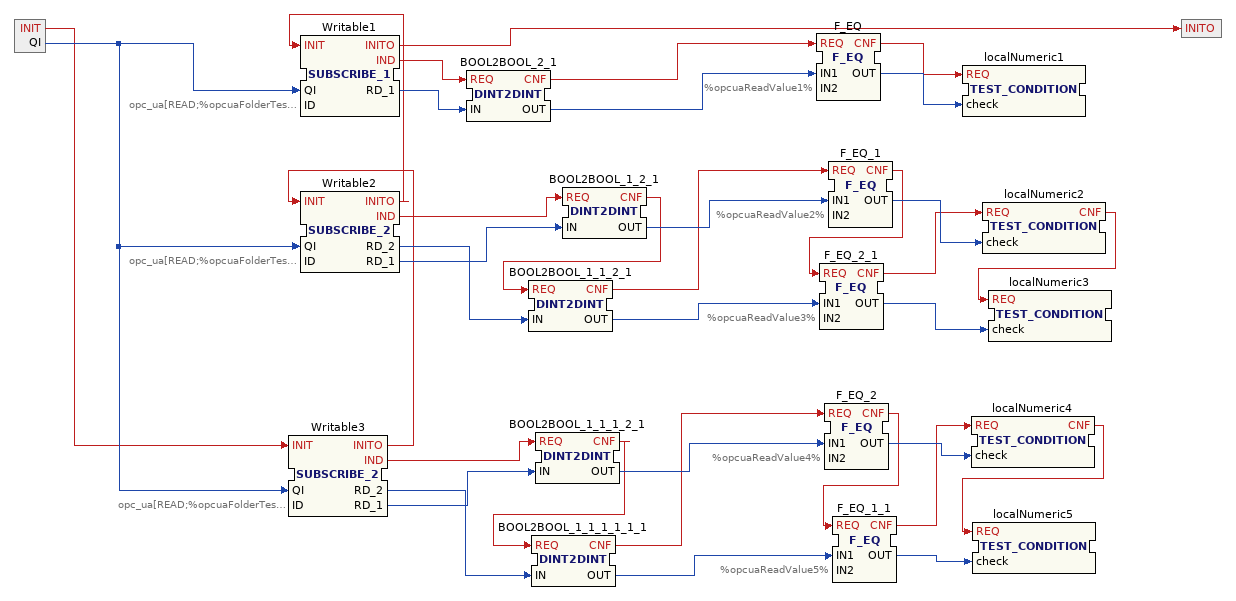
      [picture p121: application OpcUADelayedWorking.numericNodeIdTest]
      FBS
        BOOL2BOOL_1_2_1 : DINT2DINT;
        BOOL2BOOL_2_1 : DINT2DINT;
        BOOL2BOOL_1_1_2_1 : DINT2DINT;
        BOOL2BOOL_1_1_1_2_1 : DINT2DINT;
        BOOL2BOOL_1_1_1_1_1_1 : DINT2DINT;
        Writable1 : SUBSCRIBE_1(ID := opc_ua[READ;%opcuaFolderTestWithNodeIdNumeric1%]);
        Writable2 : SUBSCRIBE_2(ID := opc_ua[READ;%opcuaFolderTestWithNodeIdNumeric2%]);
        Writable3 : SUBSCRIBE_2(ID := opc_ua[READ;%opcuaFolderTestWithNodeIdNumeric3%]);
        localNumeric1 : TEST_CONDITION;
        localNumeric2 : TEST_CONDITION;
        localNumeric3 : TEST_CONDITION;
        localNumeric4 : TEST_CONDITION;
        localNumeric5 : TEST_CONDITION;
        F_EQ : F_EQ(IN2 := %opcuaReadValue1%);
        F_EQ_1 : F_EQ(IN2 := %opcuaReadValue2%);
        F_EQ_2 : F_EQ(IN2 := %opcuaReadValue4%);
        F_EQ_1_1 : F_EQ(IN2 := %opcuaReadValue5%);
        F_EQ_2_1 : F_EQ(IN2 := %opcuaReadValue3%);
      END_FBS
      EVENT_CONNECTIONS
        Writable1.INITO TO INITO;
        Writable2.INITO TO Writable1.INIT;
        INIT TO Writable3.INIT;
        Writable3.INITO TO Writable2.INIT;
        Writable1.IND TO BOOL2BOOL_2_1.REQ;
        Writable2.IND TO BOOL2BOOL_1_2_1.REQ;
        BOOL2BOOL_1_2_1.CNF TO BOOL2BOOL_1_1_2_1.REQ;
        Writable3.IND TO BOOL2BOOL_1_1_1_2_1.REQ;
        BOOL2BOOL_1_1_1_2_1.CNF TO BOOL2BOOL_1_1_1_1_1_1.REQ;
        BOOL2BOOL_2_1.CNF TO F_EQ.REQ;
        F_EQ.CNF TO localNumeric1.REQ;
        BOOL2BOOL_1_1_2_1.CNF TO F_EQ_1.REQ;
        F_EQ_1.CNF TO F_EQ_2_1.REQ;
        F_EQ_2_1.CNF TO localNumeric2.REQ;
        BOOL2BOOL_1_1_1_1_1_1.CNF TO F_EQ_2.REQ;
        F_EQ_2.CNF TO F_EQ_1_1.REQ;
        F_EQ_1_1.CNF TO localNumeric4.REQ;
        localNumeric4.CNF TO localNumeric5.REQ;
        localNumeric2.CNF TO localNumeric3.REQ;
      END_CONNECTIONS
      DATA_CONNECTIONS
        QI TO Writable1.QI;
        QI TO Writable2.QI;
        QI TO Writable3.QI;
        Writable1.RD_1 TO BOOL2BOOL_2_1.IN;
        Writable3.RD_2 TO BOOL2BOOL_1_1_1_1_1_1.IN;
        Writable3.RD_1 TO BOOL2BOOL_1_1_1_2_1.IN;
        Writable2.RD_2 TO BOOL2BOOL_1_1_2_1.IN;
        Writable2.RD_1 TO BOOL2BOOL_1_2_1.IN;
        BOOL2BOOL_2_1.OUT TO F_EQ.IN1;
        F_EQ.OUT TO localNumeric1.check;
        BOOL2BOOL_1_1_2_1.OUT TO F_EQ_2_1.IN1;
        BOOL2BOOL_1_2_1.OUT TO F_EQ_1.IN1;
        BOOL2BOOL_1_1_1_2_1.OUT TO F_EQ_2.IN1;
        BOOL2BOOL_1_1_1_1_1_1.OUT TO F_EQ_1_1.IN1;
        F_EQ_1_1.OUT TO localNumeric5.check;
        F_EQ_2.OUT TO localNumeric4.check;
        F_EQ_2_1.OUT TO localNumeric3.check;
        F_EQ_1.OUT TO localNumeric2.check;
      END_CONNECTIONS
    END_SUBAPPLICATION
    SUBAPPLICATION folderTest
      EVENT_INPUT
        INIT;
      END_EVENT
      EVENT_OUTPUT
        INITO;
      END_EVENT
      VAR_INPUT
        QI : BOOL;
      END_VAR
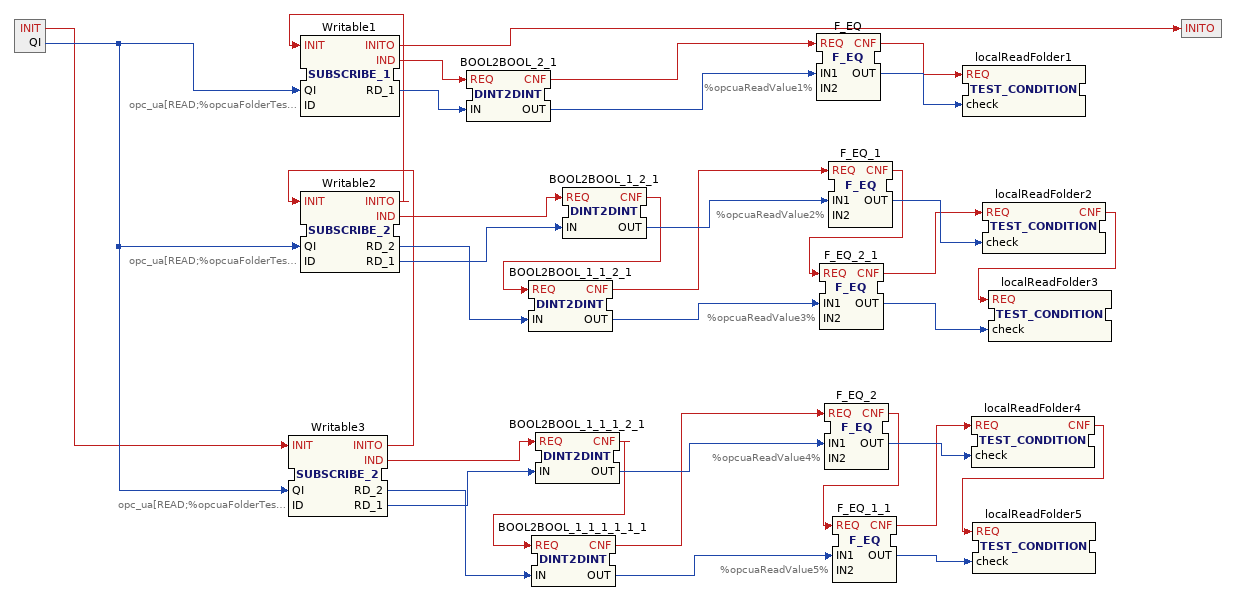
      FBS
        BOOL2BOOL_1_2_1 : DINT2DINT;
        BOOL2BOOL_2_1 : DINT2DINT;
        BOOL2BOOL_1_1_2_1 : DINT2DINT;
        BOOL2BOOL_1_1_1_2_1 : DINT2DINT;
        BOOL2BOOL_1_1_1_1_1_1 : DINT2DINT;
        Writable1 : SUBSCRIBE_1(ID := opc_ua[READ;%opcuaFolderTestOnlyBroseName1%]);
        Writable2 : SUBSCRIBE_2(ID := opc_ua[READ;%opcuaFolderTestOnlyBroseName2%]);
        Writable3 : SUBSCRIBE_2(ID := opc_ua[READ;%opcuaFolderTestOnlyBroseName3%]);
        localReadFolder1 : TEST_CONDITION;
        localReadFolder2 : TEST_CONDITION;
        localReadFolder3 : TEST_CONDITION;
        localReadFolder4 : TEST_CONDITION;
        localReadFolder5 : TEST_CONDITION;
        F_EQ : F_EQ(IN2 := %opcuaReadValue1%);
        F_EQ_1 : F_EQ(IN2 := %opcuaReadValue2%);
        F_EQ_2 : F_EQ(IN2 := %opcuaReadValue4%);
        F_EQ_1_1 : F_EQ(IN2 := %opcuaReadValue5%);
        F_EQ_2_1 : F_EQ(IN2 := %opcuaReadValue3%);
      END_FBS
      EVENT_CONNECTIONS
        Writable1.INITO TO INITO;
        Writable2.INITO TO Writable1.INIT;
        INIT TO Writable3.INIT;
        Writable3.INITO TO Writable2.INIT;
        Writable1.IND TO BOOL2BOOL_2_1.REQ;
        Writable2.IND TO BOOL2BOOL_1_2_1.REQ;
        BOOL2BOOL_1_2_1.CNF TO BOOL2BOOL_1_1_2_1.REQ;
        Writable3.IND TO BOOL2BOOL_1_1_1_2_1.REQ;
        BOOL2BOOL_1_1_1_2_1.CNF TO BOOL2BOOL_1_1_1_1_1_1.REQ;
        BOOL2BOOL_2_1.CNF TO F_EQ.REQ;
        F_EQ.CNF TO localReadFolder1.REQ;
        BOOL2BOOL_1_1_2_1.CNF TO F_EQ_1.REQ;
        F_EQ_1.CNF TO F_EQ_2_1.REQ;
        F_EQ_2_1.CNF TO localReadFolder2.REQ;
        BOOL2BOOL_1_1_1_1_1_1.CNF TO F_EQ_2.REQ;
        F_EQ_2.CNF TO F_EQ_1_1.REQ;
        F_EQ_1_1.CNF TO localReadFolder4.REQ;
        localReadFolder4.CNF TO localReadFolder5.REQ;
        localReadFolder2.CNF TO localReadFolder3.REQ;
      END_CONNECTIONS
      DATA_CONNECTIONS
        QI TO Writable1.QI;
        QI TO Writable2.QI;
        QI TO Writable3.QI;
        Writable1.RD_1 TO BOOL2BOOL_2_1.IN;
        Writable3.RD_2 TO BOOL2BOOL_1_1_1_1_1_1.IN;
        Writable3.RD_1 TO BOOL2BOOL_1_1_1_2_1.IN;
        Writable2.RD_2 TO BOOL2BOOL_1_1_2_1.IN;
        Writable2.RD_1 TO BOOL2BOOL_1_2_1.IN;
        BOOL2BOOL_2_1.OUT TO F_EQ.IN1;
        F_EQ.OUT TO localReadFolder1.check;
        BOOL2BOOL_1_1_2_1.OUT TO F_EQ_2_1.IN1;
        BOOL2BOOL_1_2_1.OUT TO F_EQ_1.IN1;
        BOOL2BOOL_1_1_1_2_1.OUT TO F_EQ_2.IN1;
        BOOL2BOOL_1_1_1_1_1_1.OUT TO F_EQ_1_1.IN1;
        F_EQ_1_1.OUT TO localReadFolder5.check;
        F_EQ_2.OUT TO localReadFolder4.check;
        F_EQ_2_1.OUT TO localReadFolder3.check;
        F_EQ_1.OUT TO localReadFolder2.check;
      END_CONNECTIONS
    END_SUBAPPLICATION
    SUBAPPLICATION byteStringNodeIdTest
      EVENT_INPUT
        INIT;
      END_EVENT
      EVENT_OUTPUT
        INITO;
      END_EVENT
      VAR_INPUT
        QI : BOOL;
      END_VAR
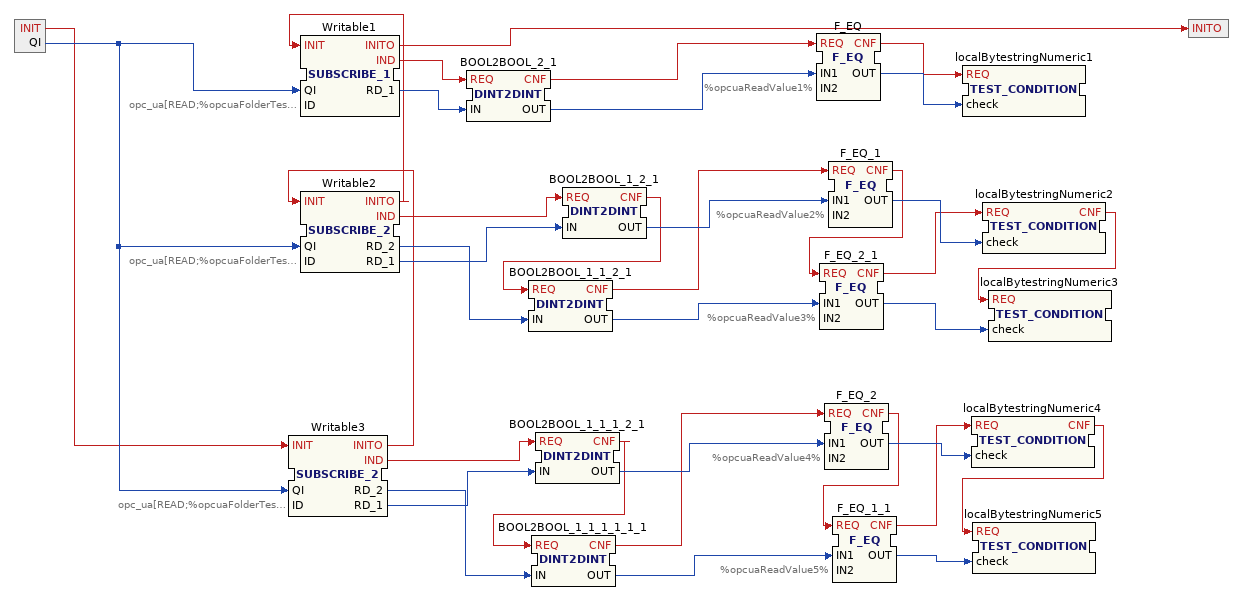
      FBS
        BOOL2BOOL_1_2_1 : DINT2DINT;
        BOOL2BOOL_2_1 : DINT2DINT;
        BOOL2BOOL_1_1_2_1 : DINT2DINT;
        BOOL2BOOL_1_1_1_2_1 : DINT2DINT;
        BOOL2BOOL_1_1_1_1_1_1 : DINT2DINT;
        Writable1 : SUBSCRIBE_1(ID := opc_ua[READ;%opcuaFolderTestWithNodeIdByteString1%]);
        Writable2 : SUBSCRIBE_2(ID := opc_ua[READ;%opcuaFolderTestWithNodeIdByteString2%]);
        Writable3 : SUBSCRIBE_2(ID := opc_ua[READ;%opcuaFolderTestWithNodeIdByteString3%]);
        localBytestringNumeric1 : TEST_CONDITION;
        localBytestringNumeric2 : TEST_CONDITION;
        localBytestringNumeric3 : TEST_CONDITION;
        localBytestringNumeric4 : TEST_CONDITION;
        localBytestringNumeric5 : TEST_CONDITION;
        F_EQ : F_EQ(IN2 := %opcuaReadValue1%);
        F_EQ_1 : F_EQ(IN2 := %opcuaReadValue2%);
        F_EQ_2 : F_EQ(IN2 := %opcuaReadValue4%);
        F_EQ_1_1 : F_EQ(IN2 := %opcuaReadValue5%);
        F_EQ_2_1 : F_EQ(IN2 := %opcuaReadValue3%);
      END_FBS
      EVENT_CONNECTIONS
        Writable1.INITO TO INITO;
        Writable2.INITO TO Writable1.INIT;
        INIT TO Writable3.INIT;
        Writable3.INITO TO Writable2.INIT;
        Writable1.IND TO BOOL2BOOL_2_1.REQ;
        Writable2.IND TO BOOL2BOOL_1_2_1.REQ;
        BOOL2BOOL_1_2_1.CNF TO BOOL2BOOL_1_1_2_1.REQ;
        Writable3.IND TO BOOL2BOOL_1_1_1_2_1.REQ;
        BOOL2BOOL_1_1_1_2_1.CNF TO BOOL2BOOL_1_1_1_1_1_1.REQ;
        BOOL2BOOL_2_1.CNF TO F_EQ.REQ;
        F_EQ.CNF TO localBytestringNumeric1.REQ;
        BOOL2BOOL_1_1_2_1.CNF TO F_EQ_1.REQ;
        F_EQ_1.CNF TO F_EQ_2_1.REQ;
        F_EQ_2_1.CNF TO localBytestringNumeric2.REQ;
        BOOL2BOOL_1_1_1_1_1_1.CNF TO F_EQ_2.REQ;
        F_EQ_2.CNF TO F_EQ_1_1.REQ;
        F_EQ_1_1.CNF TO localBytestringNumeric4.REQ;
        localBytestringNumeric4.CNF TO localBytestringNumeric5.REQ;
        localBytestringNumeric2.CNF TO localBytestringNumeric3.REQ;
      END_CONNECTIONS
      DATA_CONNECTIONS
        QI TO Writable1.QI;
        QI TO Writable2.QI;
        QI TO Writable3.QI;
        Writable1.RD_1 TO BOOL2BOOL_2_1.IN;
        Writable3.RD_2 TO BOOL2BOOL_1_1_1_1_1_1.IN;
        Writable3.RD_1 TO BOOL2BOOL_1_1_1_2_1.IN;
        Writable2.RD_2 TO BOOL2BOOL_1_1_2_1.IN;
        Writable2.RD_1 TO BOOL2BOOL_1_2_1.IN;
        BOOL2BOOL_2_1.OUT TO F_EQ.IN1;
        F_EQ.OUT TO localBytestringNumeric1.check;
        BOOL2BOOL_1_1_2_1.OUT TO F_EQ_2_1.IN1;
        BOOL2BOOL_1_2_1.OUT TO F_EQ_1.IN1;
        BOOL2BOOL_1_1_1_2_1.OUT TO F_EQ_2.IN1;
        BOOL2BOOL_1_1_1_1_1_1.OUT TO F_EQ_1_1.IN1;
        F_EQ_1_1.OUT TO localBytestringNumeric5.check;
        F_EQ_2.OUT TO localBytestringNumeric4.check;
        F_EQ_2_1.OUT TO localBytestringNumeric3.check;
        F_EQ_1.OUT TO localBytestringNumeric2.check;
      END_CONNECTIONS
    END_SUBAPPLICATION
    SUBAPPLICATION stringNodeIdTestt
      EVENT_INPUT
        INIT;
      END_EVENT
      EVENT_OUTPUT
        INITO;
      END_EVENT
      VAR_INPUT
        QI : BOOL;
      END_VAR
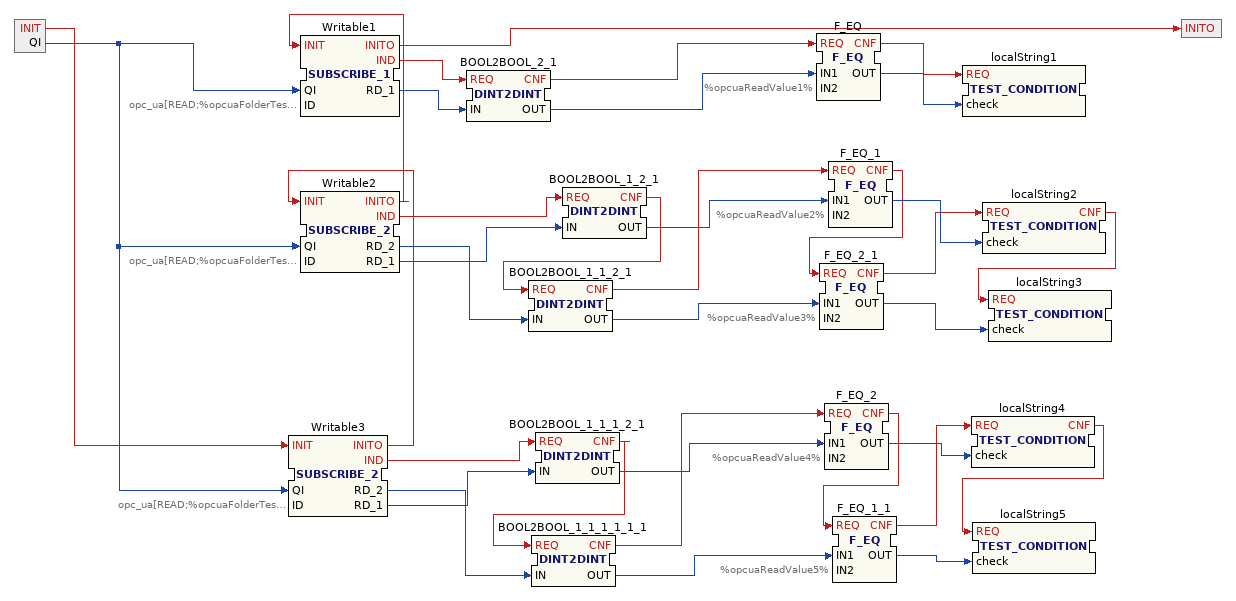
      FBS
        BOOL2BOOL_1_2_1 : DINT2DINT;
        BOOL2BOOL_2_1 : DINT2DINT;
        BOOL2BOOL_1_1_2_1 : DINT2DINT;
        BOOL2BOOL_1_1_1_2_1 : DINT2DINT;
        BOOL2BOOL_1_1_1_1_1_1 : DINT2DINT;
        Writable1 : SUBSCRIBE_1(ID := opc_ua[READ;%opcuaFolderTestWithNodeIdString1%]);
        Writable2 : SUBSCRIBE_2(ID := opc_ua[READ;%opcuaFolderTestWithNodeIdString2%]);
        Writable3 : SUBSCRIBE_2(ID := opc_ua[READ;%opcuaFolderTestWithNodeIdString3%]);
        localString1 : TEST_CONDITION;
        localString2 : TEST_CONDITION;
        localString3 : TEST_CONDITION;
        localString4 : TEST_CONDITION;
        localString5 : TEST_CONDITION;
        F_EQ : F_EQ(IN2 := %opcuaReadValue1%);
        F_EQ_1 : F_EQ(IN2 := %opcuaReadValue2%);
        F_EQ_2 : F_EQ(IN2 := %opcuaReadValue4%);
        F_EQ_1_1 : F_EQ(IN2 := %opcuaReadValue5%);
        F_EQ_2_1 : F_EQ(IN2 := %opcuaReadValue3%);
      END_FBS
      EVENT_CONNECTIONS
        Writable1.INITO TO INITO;
        Writable2.INITO TO Writable1.INIT;
        INIT TO Writable3.INIT;
        Writable3.INITO TO Writable2.INIT;
        Writable1.IND TO BOOL2BOOL_2_1.REQ;
        Writable2.IND TO BOOL2BOOL_1_2_1.REQ;
        BOOL2BOOL_1_2_1.CNF TO BOOL2BOOL_1_1_2_1.REQ;
        Writable3.IND TO BOOL2BOOL_1_1_1_2_1.REQ;
        BOOL2BOOL_1_1_1_2_1.CNF TO BOOL2BOOL_1_1_1_1_1_1.REQ;
        BOOL2BOOL_2_1.CNF TO F_EQ.REQ;
        F_EQ.CNF TO localString1.REQ;
        BOOL2BOOL_1_1_2_1.CNF TO F_EQ_1.REQ;
        F_EQ_1.CNF TO F_EQ_2_1.REQ;
        F_EQ_2_1.CNF TO localString2.REQ;
        BOOL2BOOL_1_1_1_1_1_1.CNF TO F_EQ_2.REQ;
        F_EQ_2.CNF TO F_EQ_1_1.REQ;
        F_EQ_1_1.CNF TO localString4.REQ;
        localString4.CNF TO localString5.REQ;
        localString2.CNF TO localString3.REQ;
      END_CONNECTIONS
      DATA_CONNECTIONS
        QI TO Writable1.QI;
        QI TO Writable2.QI;
        QI TO Writable3.QI;
        Writable1.RD_1 TO BOOL2BOOL_2_1.IN;
        Writable3.RD_2 TO BOOL2BOOL_1_1_1_1_1_1.IN;
        Writable3.RD_1 TO BOOL2BOOL_1_1_1_2_1.IN;
        Writable2.RD_2 TO BOOL2BOOL_1_1_2_1.IN;
        Writable2.RD_1 TO BOOL2BOOL_1_2_1.IN;
        BOOL2BOOL_2_1.OUT TO F_EQ.IN1;
        F_EQ.OUT TO localString1.check;
        BOOL2BOOL_1_1_2_1.OUT TO F_EQ_2_1.IN1;
        BOOL2BOOL_1_2_1.OUT TO F_EQ_1.IN1;
        BOOL2BOOL_1_1_1_2_1.OUT TO F_EQ_2.IN1;
        BOOL2BOOL_1_1_1_1_1_1.OUT TO F_EQ_1_1.IN1;
        F_EQ_1_1.OUT TO localString5.check;
        F_EQ_2.OUT TO localString4.check;
        F_EQ_2_1.OUT TO localString3.check;
        F_EQ_1.OUT TO localString2.check;
      END_CONNECTIONS
    END_SUBAPPLICATION
    EVENT_CONNECTIONS
      bytestringNodeIdTestRemote.INITO TO RemoteMethods.INIT;
      RemoteMethods.INITO TO HandleInit.InitFinished;
      folderTestRemote.CNF TO numericNodeIdTestRemote.REQ;
      HandleInit.Execute TO E_DELAY.START;
      SUBSCRIBE_0_1.IND TO E_SR.R;
      E_PERMIT.EO TO E_SR_1.S;
      numericNodeIdTestRemote.INITO TO stringNodeIdTestRemote.INIT;
      InitFinishedSignal.IND TO PUBLISH_0.REQ;
      E_DELAY.EO TO folderTestRemote.REQ;
      stringNodeIdTestRemote.INITO TO bytestringNodeIdTestRemote.INIT;
      bytestringNodeIdTestRemote.CNF TO RemoteMethods.REQ;
      folderTestRemote.INITO TO numericNodeIdTestRemote.INIT;
      InitFinishedSignal.INITO TO PUBLISH_0.INIT;
      numericNodeIdTestRemote.CNF TO stringNodeIdTestRemote.REQ;
      PUBLISH_0.CNF TO E_SR_2.S;
      E_SR_2.EO TO E_PERMIT.EI;
      RemoteMethods.CNF TO E_SR_1.R;
      SUBSCRIBE_0_1.INITO TO E_SR.S;
      stringNodeIdTestRemote.CNF TO bytestringNodeIdTestRemote.REQ;
      E_SR_1.EO TO folderTestRemote.INIT;
      E_SR.EO TO E_SWITCH.EI;
      E_SWITCH.EO1 TO E_SPLIT.EI;
      E_SPLIT.EO2 TO HandleInitLocal.InitFinished;
      E_SPLIT.EO1 TO E_DELAY_1.START;
      F_NOT.CNF TO E_PERMIT_1.EI;
      E_PERMIT_1.EO TO HandleInitLocal.InitFinished;
      LocaMethods.INITO TO F_NOT.REQ;
      numericNodeIdTest.INITO TO stringNodeIdTestt.INIT;
      stringNodeIdTestt.INITO TO byteStringNodeIdTest.INIT;
      folderTest.INITO TO E_DELAY_1_1.START;
      byteStringNodeIdTest.INITO TO LocaMethods.INIT;
      E_SWITCH.EO0 TO folderTest.INIT;
      E_DELAY_1.EO TO folderTest.INIT;
      E_DELAY_1_1.EO TO numericNodeIdTest.INIT;
    END_CONNECTIONS
    DATA_CONNECTIONS
      E_SR_1.Q TO RemoteMethods.QI;
      E_SR_2.Q TO E_PERMIT.PERMIT;
      E_SR_1.Q TO bytestringNodeIdTestRemote.QI;
      E_SR_1.Q TO stringNodeIdTestRemote.QI;
      E_SR.Q TO LocaMethods.QI;
      E_SR_1.Q TO folderTestRemote.QI;
      E_SR_1.Q TO numericNodeIdTestRemote.QI;
      E_SR.Q TO LocaMethods.QI;
      E_SR_1.Q TO RemoteMethods.QI;
      E_SR_1.Q TO bytestringNodeIdTestRemote.QI;
      E_SR_1.Q TO stringNodeIdTestRemote.QI;
      E_SR_1.Q TO numericNodeIdTestRemote.QI;
      E_SR_1.Q TO folderTestRemote.QI;
      E_SR.Q TO E_SWITCH.G;
      E_SR.Q TO F_NOT.IN;
      F_NOT.OUT TO E_PERMIT_1.PERMIT;
      E_SR.Q TO HandleInitLocal.QI;
      E_SR_1.Q TO HandleInit.QI;
      E_SR.Q TO folderTest.QI;
      E_SR.Q TO stringNodeIdTestt.QI;
      E_SR.Q TO byteStringNodeIdTest.QI;
      E_SR.Q TO numericNodeIdTest.QI;
    END_CONNECTIONS
  END_APPLICATION
  APPLICATION OpcUaTypes
    FBS
      Read : SUBSCRIBE_21(ID := opc_ua[READ;%opcuaTypeAll%]);
      LocalWrite : PUBLISH_21(ID := opc_ua[WRITE;%opcuaTypeAll%]);
      RemoteCall : CLIENT_21(ID := opc_ua[%callMethodAction%;%serverEndpoint%;%opcuaTypeNode%]);
      Method : SERVER_21(ID := opc_ua[CREATE_METHOD;%opcuaTypeNode%]);
      E_SR : E_SR;
      SUBSCRIBE_0_1 : SUBSCRIBE_0(QI := 1, ID := %clientEnded%);
      E_SWITCH : E_SWITCH;
      E_DELAY : E_DELAY(DT := T#1500ms);
      E_SR_1 : E_SR;
      E_SR_2 : E_SR;
      PUBLISH_0 : PUBLISH_0(QI := 1, ID := %serverInitCommIdACK%);
      E_PERMIT : E_PERMIT;
      InitFinishedSignal : SUBSCRIBE_0(QI := 1, ID := %serverInitCommId%);
      RemoteRead : CLIENT_0_21(ID := opc_ua[READ;%serverEndpoint%;%opcuaTypeAll%]);
      RemoteWrite : CLIENT_21_0(ID := opc_ua[WRITE;%serverEndpoint%;%opcuaTypeAll%]);
      RemoteWriteAll : TEST_CONDITION;
    END_FBS
    SUBAPPLICATION AllTypes
      EVENT_INPUT
        REQ;
      END_EVENT
      EVENT_OUTPUT
        CNF;
      END_EVENT
      VAR_INPUT
        BOOL_I : BOOL; (* BOOL Type Input *)
        SINT_I : SINT; (* SINT Type Input *)
        INT_I : INT; (* INT Type Input *)
        DINT_I : DINT; (* DINT Type Input *)
        LINT_I : LINT; (* LINT Type Input *)
        USINT_I : USINT; (* USINT Type Input *)
        UINT_I : UINT; (* UINT Type Input *)
        UDINT_I : UDINT; (* UDINT Type Input *)
        ULINT_I : ULINT; (* ULINT Type Input *)
        BYTE_I : BYTE; (* BYTE Type Input *)
        WORD_I : WORD; (* WORD Type Input *)
        DWORD_I : DWORD; (* DWORD Type Input *)
        LWORD_I : LWORD; (* LWORD Type Input *)
        DATE_I_BOOL : BOOL; (* DATE Type Input *)
        TIME_OF_DAY_I_BOOL : BOOL; (* TIME_OF_DAY Type Input *)
        DATE_AND_TIME_I_BOOL : BOOL; (* DATE_AND_TIME Type Input *)
        TIME_I : TIME; (* TIME Type Input *)
        REAL_I : REAL; (* REAL Type Input *)
        LREAL_I : LREAL; (* LREAL Type Input *)
        STRING_I : STRING; (* STRING Type Input *)
        WSTRING_I : WSTRING; (* WSTRING Type Input *)
      END_VAR
      VAR_OUTPUT
        BOOL_O : BOOL; (* BOOL Type Output *)
        SINT_O : SINT; (* SINT Type Output *)
        INT_O : INT; (* INT Type Output *)
        DINT_O : DINT; (* DINT Type Output *)
        LINT_O : LINT; (* LINT Type Output *)
        USINT_O : USINT; (* USINT Type Output *)
        UINT_O : UINT; (* UINT Type Output *)
        UDINT_O : UDINT; (* UDINT Type Output *)
        ULINT_O : ULINT; (* ULINT Type Output *)
        BYTE_O : BYTE; (* BYTE Type Output *)
        WORD_O : WORD; (* WORD Type Output *)
        DWORD_O : DWORD; (* DWORD Type Output *)
        LWORD_O : LWORD; (* LWORD Type Output *)
        DATE_O_BOOL : BOOL; (* DATE Type Output *)
        TIME_OF_DAY_O_BOOL : BOOL; (* TIME_OF_DAY Type Output *)
        DATE_AND_TIME_O_BOOL : BOOL; (* DATE_AND_TIME Type Output *)
        TIME_O : TIME; (* TIME Type Output *)
        REAL_O : REAL; (* REAL Type Output *)
        LREAL_O : LREAL; (* LREAL Type Output *)
        STRING_O : STRING; (* STRING Type Output *)
        WSTRING_O : WSTRING; (* WSTRING Type Output *)
      END_VAR
      FBS
        SINT2SINT : SINT2SINT;
        UINT2UINT : UINT2UINT;
        BOOL2BOOL : BOOL2BOOL;
        UDINT2UDINT : UDINT2UDINT;
        DINT2DINT : DINT2DINT;
        F_LINT_TO_INT : F_LINT_TO_INT;
        INT2INT : INT2INT;
        USINT2USINT : USINT2USINT;
        F_ULINT_TO_INT : F_ULINT_TO_INT;
        BYTE2BYTE : BYTE2BYTE;
        WORD2WORD : WORD2WORD;
        DWORD2DWORD : DWORD2DWORD;
        F_LWORD_TO_INT : F_LWORD_TO_INT;
        MISSING_DATE : F_DT_TO_DATE;
        MISSING_DATE_AND_TIME : F_DT_TO_TOD;
        TIME2TIME : TIME2TIME;
        REAL2REAL : REAL2REAL;
        LREAL2LREAL : LREAL2LREAL;
        STRING2STRING : STRING2STRING;
        WSTRING2WSTRING : WSTRING2WSTRING;
        Time_of_day : F_ADD_TOD_TIME;
        F_INT_TO_LINT : F_INT_TO_LINT;
        F_INT_TO_ULINT : F_INT_TO_ULINT;
        F_INT_TO_LWORD : F_INT_TO_LWORD;
        BOOL2BOOL_1 : BOOL2BOOL;
        BOOL2BOOL_2 : BOOL2BOOL;
        BOOL2BOOL_3 : BOOL2BOOL;
      END_FBS
      EVENT_CONNECTIONS
        REQ TO BOOL2BOOL.REQ;
        F_LINT_TO_INT.CNF TO F_INT_TO_LINT.REQ;
        F_ULINT_TO_INT.CNF TO F_INT_TO_ULINT.REQ;
        F_LWORD_TO_INT.CNF TO F_INT_TO_LWORD.REQ;
        BOOL2BOOL.CNF TO SINT2SINT.REQ;
        SINT2SINT.CNF TO INT2INT.REQ;
        INT2INT.CNF TO DINT2DINT.REQ;
        DINT2DINT.CNF TO F_LINT_TO_INT.REQ;
        F_INT_TO_LINT.CNF TO USINT2USINT.REQ;
        USINT2USINT.CNF TO UINT2UINT.REQ;
        UINT2UINT.CNF TO UDINT2UDINT.REQ;
        UDINT2UDINT.CNF TO F_ULINT_TO_INT.REQ;
        F_INT_TO_ULINT.CNF TO BYTE2BYTE.REQ;
        BYTE2BYTE.CNF TO WORD2WORD.REQ;
        WORD2WORD.CNF TO DWORD2DWORD.REQ;
        DWORD2DWORD.CNF TO F_LWORD_TO_INT.REQ;
        F_INT_TO_LWORD.CNF TO BOOL2BOOL_1.REQ;
        BOOL2BOOL_1.CNF TO BOOL2BOOL_2.REQ;
        BOOL2BOOL_2.CNF TO BOOL2BOOL_3.REQ;
        BOOL2BOOL_3.CNF TO TIME2TIME.REQ;
        TIME2TIME.CNF TO REAL2REAL.REQ;
        REAL2REAL.CNF TO LREAL2LREAL.REQ;
        LREAL2LREAL.CNF TO STRING2STRING.REQ;
        STRING2STRING.CNF TO WSTRING2WSTRING.REQ;
        WSTRING2WSTRING.CNF TO CNF;
      END_CONNECTIONS
      DATA_CONNECTIONS
        BOOL_I TO BOOL2BOOL.IN;
        SINT_I TO SINT2SINT.IN;
        INT_I TO INT2INT.IN;
        DINT_I TO DINT2DINT.IN;
        LINT_I TO F_LINT_TO_INT.IN;
        USINT_I TO USINT2USINT.IN;
        UINT_I TO UINT2UINT.IN;
        UDINT_I TO UDINT2UDINT.IN;
        ULINT_I TO F_ULINT_TO_INT.IN;
        BYTE_I TO BYTE2BYTE.IN;
        WORD_I TO WORD2WORD.IN;
        DWORD_I TO DWORD2DWORD.IN;
        LWORD_I TO F_LWORD_TO_INT.IN;
        TIME_I TO TIME2TIME.IN;
        REAL_I TO REAL2REAL.IN;
        LREAL_I TO LREAL2LREAL.IN;
        STRING_I TO STRING2STRING.IN;
        WSTRING_I TO WSTRING2WSTRING.IN;
        SINT2SINT.OUT TO SINT_O;
        INT2INT.OUT TO INT_O;
        DINT2DINT.OUT TO DINT_O;
        F_LINT_TO_INT.OUT TO F_INT_TO_LINT.IN;
        F_INT_TO_LINT.OUT TO LINT_O;
        USINT2USINT.OUT TO USINT_O;
        UINT2UINT.OUT TO UINT_O;
        UDINT2UDINT.OUT TO UDINT_O;
        F_ULINT_TO_INT.OUT TO F_INT_TO_ULINT.IN;
        F_INT_TO_ULINT.OUT TO ULINT_O;
        BYTE2BYTE.OUT TO BYTE_O;
        WORD2WORD.OUT TO WORD_O;
        DWORD2DWORD.OUT TO DWORD_O;
        F_LWORD_TO_INT.OUT TO F_INT_TO_LWORD.IN;
        F_INT_TO_LWORD.OUT TO LWORD_O;
        WSTRING2WSTRING.OUT TO WSTRING_O;
        STRING2STRING.OUT TO STRING_O;
        LREAL2LREAL.OUT TO LREAL_O;
        REAL2REAL.OUT TO REAL_O;
        TIME2TIME.OUT TO TIME_O;
        DATE_I_BOOL TO BOOL2BOOL_1.IN;
        TIME_OF_DAY_I_BOOL TO BOOL2BOOL_2.IN;
        DATE_AND_TIME_I_BOOL TO BOOL2BOOL_3.IN;
        BOOL2BOOL_1.OUT TO DATE_O_BOOL;
        BOOL2BOOL_2.OUT TO TIME_OF_DAY_O_BOOL;
        BOOL2BOOL_3.OUT TO DATE_AND_TIME_O_BOOL;
        BOOL2BOOL.OUT TO BOOL_O;
      END_CONNECTIONS
    END_SUBAPPLICATION
    SUBAPPLICATION TypeTest
      EVENT_INPUT
        REQ;
      END_EVENT
      EVENT_OUTPUT
        CNF;
      END_EVENT
      VAR_INPUT
        BOOL_I : BOOL; (* BOOL Type Input *)
        SINT_I : SINT; (* SINT Type Input *)
        INT_I : INT; (* INT Type Input *)
        DINT_I : DINT; (* DINT Type Input *)
        LINT_I : LINT; (* LINT Type Input *)
        USINT_I : USINT; (* USINT Type Input *)
        UINT_I : UINT; (* UINT Type Input *)
        UDINT_I : UDINT; (* UDINT Type Input *)
        ULINT_I : ULINT; (* ULINT Type Input *)
        BYTE_I : BYTE; (* BYTE Type Input *)
        WORD_I : WORD; (* WORD Type Input *)
        DWORD_I : DWORD; (* DWORD Type Input *)
        LWORD_I : LWORD; (* LWORD Type Input *)
        DATE_I : DATE; (* DATE Type Input *)
        TIME_OF_DAY_I : TIME_OF_DAY; (* TIME_OF_DAY Type Input *)
        DATE_AND_TIME_I : DATE_AND_TIME; (* DATE_AND_TIME Type Input *)
        TIME_I : TIME; (* TIME Type Input *)
        REAL_I : REAL; (* REAL Type Input *)
        LREAL_I : LREAL; (* LREAL Type Input *)
        STRING_I : STRING; (* STRING Type Input *)
        WSTRING_I : WSTRING; (* WSTRING Type Input *)
      END_VAR
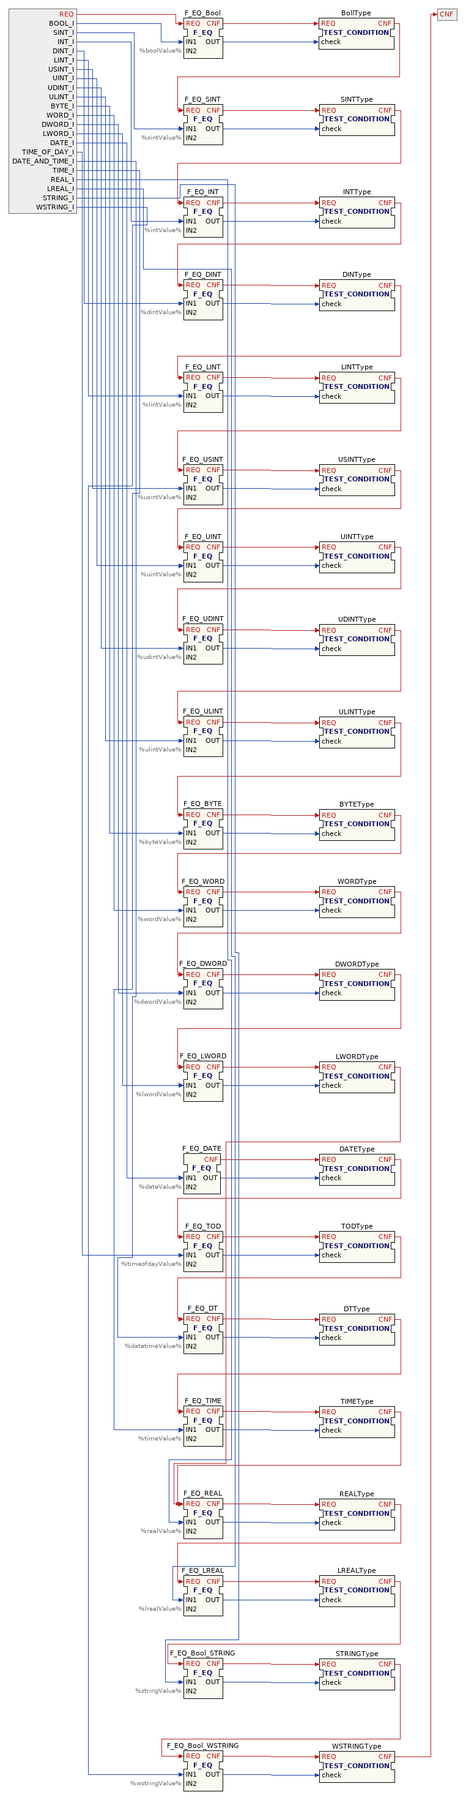
      FBS
        BollType : TEST_CONDITION;
        F_EQ_Bool : F_EQ(IN2 := %boolValue%);
        SINTType : TEST_CONDITION;
        F_EQ_SINT : F_EQ(IN2 := %sintValue%);
        INTType : TEST_CONDITION;
        F_EQ_INT : F_EQ(IN2 := %intValue%);
        DINType : TEST_CONDITION;
        F_EQ_DINT : F_EQ(IN2 := %dintValue%);
        F_EQ_USINT : F_EQ(IN2 := %usintValue%);
        USINTType : TEST_CONDITION;
        F_EQ_UINT : F_EQ(IN2 := %uintValue%);
        LINTType : TEST_CONDITION;
        UINTType : TEST_CONDITION;
        UDINTType : TEST_CONDITION;
        F_EQ_UDINT : F_EQ(IN2 := %udintValue%);
        F_EQ_LINT : F_EQ(IN2 := %lintValue%);
        F_EQ_BYTE : F_EQ(IN2 := %byteValue%);
        BYTEType : TEST_CONDITION;
        F_EQ_WORD : F_EQ(IN2 := %wordValue%);
        ULINTType : TEST_CONDITION;
        WORDType : TEST_CONDITION;
        DWORDType : TEST_CONDITION;
        F_EQ_DWORD : F_EQ(IN2 := %dwordValue%);
        F_EQ_ULINT : F_EQ(IN2 := %ulintValue%);
        F_EQ_DATE : F_EQ(IN2 := %dateValue%);
        DATEType : TEST_CONDITION;
        F_EQ_LREAL : F_EQ(IN2 := %lrealValue%);
        LWORDType : TEST_CONDITION;
        TODType : TEST_CONDITION;
        DTType : TEST_CONDITION;
        F_EQ_DT : F_EQ(IN2 := %datetimeValue%);
        REALType : TEST_CONDITION;
        LREALType : TEST_CONDITION;
        F_EQ_REAL : F_EQ(IN2 := %realValue%);
        F_EQ_LWORD : F_EQ(IN2 := %lwordValue%);
        WSTRINGType : TEST_CONDITION;
        F_EQ_TIME : F_EQ(IN2 := %timeValue%);
        STRINGType : TEST_CONDITION;
        F_EQ_TOD : F_EQ(IN2 := %timeofdayValue%);
        F_EQ_Bool_STRING : F_EQ(IN2 := %stringValue%);
        F_EQ_Bool_WSTRING : F_EQ(IN2 := %wstringValue%);
        TIMEType : TEST_CONDITION;
      END_FBS
      EVENT_CONNECTIONS
        F_EQ_Bool.CNF TO BollType.REQ;
        F_EQ_SINT.CNF TO SINTType.REQ;
        F_EQ_INT.CNF TO INTType.REQ;
        F_EQ_DINT.CNF TO DINType.REQ;
        F_EQ_UINT.CNF TO UINTType.REQ;
        F_EQ_UDINT.CNF TO UDINTType.REQ;
        F_EQ_USINT.CNF TO USINTType.REQ;
        F_EQ_LINT.CNF TO LINTType.REQ;
        F_EQ_WORD.CNF TO WORDType.REQ;
        F_EQ_DWORD.CNF TO DWORDType.REQ;
        F_EQ_BYTE.CNF TO BYTEType.REQ;
        F_EQ_ULINT.CNF TO ULINTType.REQ;
        F_EQ_REAL.CNF TO REALType.REQ;
        F_EQ_TOD.CNF TO TODType.REQ;
        F_EQ_Bool_STRING.CNF TO STRINGType.REQ;
        F_EQ_LREAL.CNF TO LREALType.REQ;
        F_EQ_DT.CNF TO DTType.REQ;
        F_EQ_Bool_WSTRING.CNF TO WSTRINGType.REQ;
        F_EQ_LWORD.CNF TO LWORDType.REQ;
        F_EQ_DATE.CNF TO DATEType.REQ;
        F_EQ_TIME.CNF TO TIMEType.REQ;
        REQ TO F_EQ_Bool.REQ;
        BollType.CNF TO F_EQ_SINT.REQ;
        SINTType.CNF TO F_EQ_INT.REQ;
        INTType.CNF TO F_EQ_DINT.REQ;
        DINType.CNF TO F_EQ_LINT.REQ;
        LINTType.CNF TO F_EQ_USINT.REQ;
        USINTType.CNF TO F_EQ_UINT.REQ;
        UINTType.CNF TO F_EQ_UDINT.REQ;
        UDINTType.CNF TO F_EQ_ULINT.REQ;
        ULINTType.CNF TO F_EQ_BYTE.REQ;
        BYTEType.CNF TO F_EQ_WORD.REQ;
        WORDType.CNF TO F_EQ_DWORD.REQ;
        DWORDType.CNF TO F_EQ_LWORD.REQ;
        DATEType.CNF TO F_EQ_TOD.REQ;
        TODType.CNF TO F_EQ_DT.REQ;
        DTType.CNF TO F_EQ_TIME.REQ;
        TIMEType.CNF TO F_EQ_REAL.REQ;
        REALType.CNF TO F_EQ_LREAL.REQ;
        LREALType.CNF TO F_EQ_Bool_STRING.REQ;
        STRINGType.CNF TO F_EQ_Bool_WSTRING.REQ;
        LWORDType.CNF TO F_EQ_REAL.REQ;
        WSTRINGType.CNF TO CNF;
      END_CONNECTIONS
      DATA_CONNECTIONS
        F_EQ_Bool.OUT TO BollType.check;
        F_EQ_SINT.OUT TO SINTType.check;
        F_EQ_INT.OUT TO INTType.check;
        F_EQ_DINT.OUT TO DINType.check;
        F_EQ_UINT.OUT TO UINTType.check;
        F_EQ_LINT.OUT TO LINTType.check;
        F_EQ_USINT.OUT TO USINTType.check;
        F_EQ_UDINT.OUT TO UDINTType.check;
        F_EQ_WORD.OUT TO WORDType.check;
        F_EQ_ULINT.OUT TO ULINTType.check;
        F_EQ_BYTE.OUT TO BYTEType.check;
        F_EQ_DWORD.OUT TO DWORDType.check;
        F_EQ_TOD.OUT TO TODType.check;
        F_EQ_LWORD.OUT TO LWORDType.check;
        F_EQ_Bool_WSTRING.OUT TO WSTRINGType.check;
        F_EQ_LREAL.OUT TO LREALType.check;
        F_EQ_DATE.OUT TO DATEType.check;
        F_EQ_Bool_STRING.OUT TO STRINGType.check;
        F_EQ_TIME.OUT TO TIMEType.check;
        F_EQ_REAL.OUT TO REALType.check;
        F_EQ_DT.OUT TO DTType.check;
        SINT_I TO F_EQ_SINT.IN1;
        INT_I TO F_EQ_INT.IN1;
        DINT_I TO F_EQ_DINT.IN1;
        LINT_I TO F_EQ_LINT.IN1;
        USINT_I TO F_EQ_USINT.IN1;
        UINT_I TO F_EQ_UINT.IN1;
        UDINT_I TO F_EQ_UDINT.IN1;
        ULINT_I TO F_EQ_ULINT.IN1;
        BYTE_I TO F_EQ_BYTE.IN1;
        WORD_I TO F_EQ_WORD.IN1;
        DWORD_I TO F_EQ_DWORD.IN1;
        LWORD_I TO F_EQ_LWORD.IN1;
        DATE_I TO F_EQ_DATE.IN1;
        TIME_OF_DAY_I TO F_EQ_TOD.IN1;
        DATE_AND_TIME_I TO F_EQ_DT.IN1;
        TIME_I TO F_EQ_TIME.IN1;
        REAL_I TO F_EQ_REAL.IN1;
        LREAL_I TO F_EQ_LREAL.IN1;
        STRING_I TO F_EQ_Bool_STRING.IN1;
        WSTRING_I TO F_EQ_Bool_WSTRING.IN1;
        BOOL_I TO F_EQ_Bool.IN1;
      END_CONNECTIONS
    END_SUBAPPLICATION
    SUBAPPLICATION AllTypes_2
      EVENT_INPUT
        REQ;
      END_EVENT
      EVENT_OUTPUT
        CNF;
      END_EVENT
      VAR_INPUT
        BOOL_I : BOOL; (* BOOL Type Input *)
        SINT_I : SINT; (* SINT Type Input *)
        INT_I : INT; (* INT Type Input *)
        DINT_I : DINT; (* DINT Type Input *)
        LINT_I : LINT; (* LINT Type Input *)
        USINT_I : USINT; (* USINT Type Input *)
        UINT_I : UINT; (* UINT Type Input *)
        UDINT_I : UDINT; (* UDINT Type Input *)
        ULINT_I : ULINT; (* ULINT Type Input *)
        BYTE_I : BYTE; (* BYTE Type Input *)
        WORD_I : WORD; (* WORD Type Input *)
        DWORD_I : DWORD; (* DWORD Type Input *)
        LWORD_I : LWORD; (* LWORD Type Input *)
        DATE_I_BOOL : BOOL; (* DATE Type Input *)
        TIME_OF_DAY_I_BOOL : BOOL; (* TIME_OF_DAY Type Input *)
        DATE_AND_TIME_I_BOOL : BOOL; (* DATE_AND_TIME Type Input *)
        TIME_I : TIME; (* TIME Type Input *)
        REAL_I : REAL; (* REAL Type Input *)
        LREAL_I : LREAL; (* LREAL Type Input *)
        STRING_I : STRING; (* STRING Type Input *)
        WSTRING_I : WSTRING; (* WSTRING Type Input *)
      END_VAR
      VAR_OUTPUT
        BOOL_O : BOOL; (* BOOL Type Output *)
        SINT_O : SINT; (* SINT Type Output *)
        INT_O : INT; (* INT Type Output *)
        DINT_O : DINT; (* DINT Type Output *)
        LINT_O : LINT; (* LINT Type Output *)
        USINT_O : USINT; (* USINT Type Output *)
        UINT_O : UINT; (* UINT Type Output *)
        UDINT_O : UDINT; (* UDINT Type Output *)
        ULINT_O : ULINT; (* ULINT Type Output *)
        BYTE_O : BYTE; (* BYTE Type Output *)
        WORD_O : WORD; (* WORD Type Output *)
        DWORD_O : DWORD; (* DWORD Type Output *)
        LWORD_O : LWORD; (* LWORD Type Output *)
        DATE_O_BOOL : BOOL; (* DATE Type Output *)
        TIME_OF_DAY_O_BOOL : BOOL; (* TIME_OF_DAY Type Output *)
        DATE_AND_TIME_O_BOOL : BOOL; (* DATE_AND_TIME Type Output *)
        TIME_O : TIME; (* TIME Type Output *)
        REAL_O : REAL; (* REAL Type Output *)
        LREAL_O : LREAL; (* LREAL Type Output *)
        STRING_O : STRING; (* STRING Type Output *)
        WSTRING_O : WSTRING; (* WSTRING Type Output *)
      END_VAR
      FBS
        SINT2SINT : SINT2SINT;
        UINT2UINT : UINT2UINT;
        BOOL2BOOL : BOOL2BOOL;
        UDINT2UDINT : UDINT2UDINT;
        DINT2DINT : DINT2DINT;
        F_LINT_TO_INT : F_LINT_TO_INT;
        INT2INT : INT2INT;
        USINT2USINT : USINT2USINT;
        F_ULINT_TO_INT : F_ULINT_TO_INT;
        BYTE2BYTE : BYTE2BYTE;
        WORD2WORD : WORD2WORD;
        DWORD2DWORD : DWORD2DWORD;
        F_LWORD_TO_INT : F_LWORD_TO_INT;
        MISSING_DATE : F_DT_TO_DATE;
        MISSING_DATE_AND_TIME : F_DT_TO_TOD;
        TIME2TIME : TIME2TIME;
        REAL2REAL : REAL2REAL;
        LREAL2LREAL : LREAL2LREAL;
        STRING2STRING : STRING2STRING;
        WSTRING2WSTRING : WSTRING2WSTRING;
        Time_of_day : F_ADD_TOD_TIME;
        F_INT_TO_LINT : F_INT_TO_LINT;
        F_INT_TO_ULINT : F_INT_TO_ULINT;
        F_INT_TO_LWORD : F_INT_TO_LWORD;
        BOOL2BOOL_1 : BOOL2BOOL;
        BOOL2BOOL_2 : BOOL2BOOL;
        BOOL2BOOL_3 : BOOL2BOOL;
      END_FBS
      EVENT_CONNECTIONS
        REQ TO BOOL2BOOL.REQ;
        F_LINT_TO_INT.CNF TO F_INT_TO_LINT.REQ;
        F_ULINT_TO_INT.CNF TO F_INT_TO_ULINT.REQ;
        F_LWORD_TO_INT.CNF TO F_INT_TO_LWORD.REQ;
        BOOL2BOOL.CNF TO SINT2SINT.REQ;
        SINT2SINT.CNF TO INT2INT.REQ;
        INT2INT.CNF TO DINT2DINT.REQ;
        DINT2DINT.CNF TO F_LINT_TO_INT.REQ;
        F_INT_TO_LINT.CNF TO USINT2USINT.REQ;
        USINT2USINT.CNF TO UINT2UINT.REQ;
        UINT2UINT.CNF TO UDINT2UDINT.REQ;
        UDINT2UDINT.CNF TO F_ULINT_TO_INT.REQ;
        F_INT_TO_ULINT.CNF TO BYTE2BYTE.REQ;
        BYTE2BYTE.CNF TO WORD2WORD.REQ;
        WORD2WORD.CNF TO DWORD2DWORD.REQ;
        DWORD2DWORD.CNF TO F_LWORD_TO_INT.REQ;
        F_INT_TO_LWORD.CNF TO BOOL2BOOL_1.REQ;
        BOOL2BOOL_1.CNF TO BOOL2BOOL_2.REQ;
        BOOL2BOOL_2.CNF TO BOOL2BOOL_3.REQ;
        BOOL2BOOL_3.CNF TO TIME2TIME.REQ;
        TIME2TIME.CNF TO REAL2REAL.REQ;
        REAL2REAL.CNF TO LREAL2LREAL.REQ;
        LREAL2LREAL.CNF TO STRING2STRING.REQ;
        STRING2STRING.CNF TO WSTRING2WSTRING.REQ;
        WSTRING2WSTRING.CNF TO CNF;
      END_CONNECTIONS
      DATA_CONNECTIONS
        BOOL_I TO BOOL2BOOL.IN;
        SINT_I TO SINT2SINT.IN;
        INT_I TO INT2INT.IN;
        DINT_I TO DINT2DINT.IN;
        LINT_I TO F_LINT_TO_INT.IN;
        USINT_I TO USINT2USINT.IN;
        UINT_I TO UINT2UINT.IN;
        UDINT_I TO UDINT2UDINT.IN;
        ULINT_I TO F_ULINT_TO_INT.IN;
        BYTE_I TO BYTE2BYTE.IN;
        WORD_I TO WORD2WORD.IN;
        DWORD_I TO DWORD2DWORD.IN;
        LWORD_I TO F_LWORD_TO_INT.IN;
        TIME_I TO TIME2TIME.IN;
        REAL_I TO REAL2REAL.IN;
        LREAL_I TO LREAL2LREAL.IN;
        STRING_I TO STRING2STRING.IN;
        WSTRING_I TO WSTRING2WSTRING.IN;
        SINT2SINT.OUT TO SINT_O;
        INT2INT.OUT TO INT_O;
        DINT2DINT.OUT TO DINT_O;
        F_LINT_TO_INT.OUT TO F_INT_TO_LINT.IN;
        F_INT_TO_LINT.OUT TO LINT_O;
        USINT2USINT.OUT TO USINT_O;
        UINT2UINT.OUT TO UINT_O;
        UDINT2UDINT.OUT TO UDINT_O;
        F_ULINT_TO_INT.OUT TO F_INT_TO_ULINT.IN;
        F_INT_TO_ULINT.OUT TO ULINT_O;
        BYTE2BYTE.OUT TO BYTE_O;
        WORD2WORD.OUT TO WORD_O;
        DWORD2DWORD.OUT TO DWORD_O;
        F_LWORD_TO_INT.OUT TO F_INT_TO_LWORD.IN;
        F_INT_TO_LWORD.OUT TO LWORD_O;
        WSTRING2WSTRING.OUT TO WSTRING_O;
        STRING2STRING.OUT TO STRING_O;
        LREAL2LREAL.OUT TO LREAL_O;
        REAL2REAL.OUT TO REAL_O;
        TIME2TIME.OUT TO TIME_O;
        DATE_I_BOOL TO BOOL2BOOL_1.IN;
        TIME_OF_DAY_I_BOOL TO BOOL2BOOL_2.IN;
        DATE_AND_TIME_I_BOOL TO BOOL2BOOL_3.IN;
        BOOL2BOOL_1.OUT TO DATE_O_BOOL;
        BOOL2BOOL_2.OUT TO TIME_OF_DAY_O_BOOL;
        BOOL2BOOL_3.OUT TO DATE_AND_TIME_O_BOOL;
        BOOL2BOOL.OUT TO BOOL_O;
      END_CONNECTIONS
    END_SUBAPPLICATION
    SUBAPPLICATION TypeTest_1
      EVENT_INPUT
        REQ;
      END_EVENT
      EVENT_OUTPUT
        CNF;
      END_EVENT
      VAR_INPUT
        BOOL_I : BOOL; (* BOOL Type Input *)
        SINT_I : SINT; (* SINT Type Input *)
        INT_I : INT; (* INT Type Input *)
        DINT_I : DINT; (* DINT Type Input *)
        LINT_I : LINT; (* LINT Type Input *)
        USINT_I : USINT; (* USINT Type Input *)
        UINT_I : UINT; (* UINT Type Input *)
        UDINT_I : UDINT; (* UDINT Type Input *)
        ULINT_I : ULINT; (* ULINT Type Input *)
        BYTE_I : BYTE; (* BYTE Type Input *)
        WORD_I : WORD; (* WORD Type Input *)
        DWORD_I : DWORD; (* DWORD Type Input *)
        LWORD_I : LWORD; (* LWORD Type Input *)
        DATE_I : DATE; (* DATE Type Input *)
        TIME_OF_DAY_I : TIME_OF_DAY; (* TIME_OF_DAY Type Input *)
        DATE_AND_TIME_I : DATE_AND_TIME; (* DATE_AND_TIME Type Input *)
        TIME_I : TIME; (* TIME Type Input *)
        REAL_I : REAL; (* REAL Type Input *)
        LREAL_I : LREAL; (* LREAL Type Input *)
        STRING_I : STRING; (* STRING Type Input *)
        WSTRING_I : WSTRING; (* WSTRING Type Input *)
      END_VAR
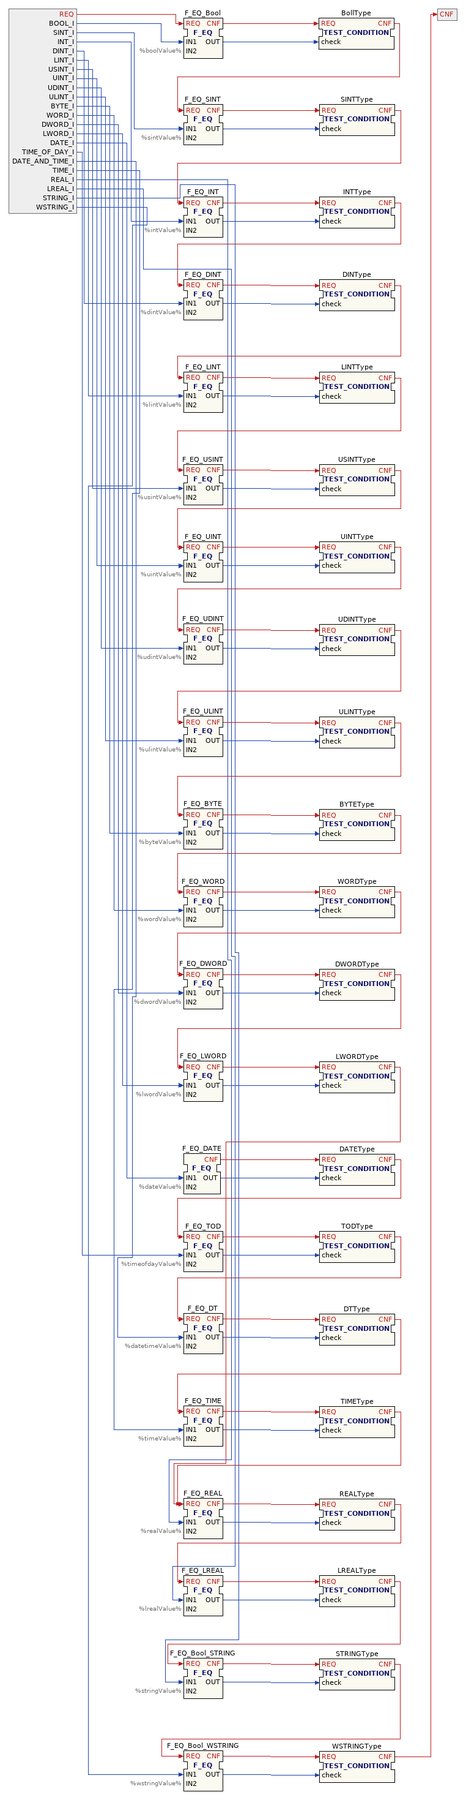
      FBS
        BollType : TEST_CONDITION;
        F_EQ_Bool : F_EQ(IN2 := %boolValue%);
        SINTType : TEST_CONDITION;
        F_EQ_SINT : F_EQ(IN2 := %sintValue%);
        INTType : TEST_CONDITION;
        F_EQ_INT : F_EQ(IN2 := %intValue%);
        DINType : TEST_CONDITION;
        F_EQ_DINT : F_EQ(IN2 := %dintValue%);
        F_EQ_USINT : F_EQ(IN2 := %usintValue%);
        USINTType : TEST_CONDITION;
        F_EQ_UINT : F_EQ(IN2 := %uintValue%);
        LINTType : TEST_CONDITION;
        UINTType : TEST_CONDITION;
        UDINTType : TEST_CONDITION;
        F_EQ_UDINT : F_EQ(IN2 := %udintValue%);
        F_EQ_LINT : F_EQ(IN2 := %lintValue%);
        F_EQ_BYTE : F_EQ(IN2 := %byteValue%);
        BYTEType : TEST_CONDITION;
        F_EQ_WORD : F_EQ(IN2 := %wordValue%);
        ULINTType : TEST_CONDITION;
        WORDType : TEST_CONDITION;
        DWORDType : TEST_CONDITION;
        F_EQ_DWORD : F_EQ(IN2 := %dwordValue%);
        F_EQ_ULINT : F_EQ(IN2 := %ulintValue%);
        F_EQ_DATE : F_EQ(IN2 := %dateValue%);
        DATEType : TEST_CONDITION;
        F_EQ_LREAL : F_EQ(IN2 := %lrealValue%);
        LWORDType : TEST_CONDITION;
        TODType : TEST_CONDITION;
        DTType : TEST_CONDITION;
        F_EQ_DT : F_EQ(IN2 := %datetimeValue%);
        REALType : TEST_CONDITION;
        LREALType : TEST_CONDITION;
        F_EQ_REAL : F_EQ(IN2 := %realValue%);
        F_EQ_LWORD : F_EQ(IN2 := %lwordValue%);
        WSTRINGType : TEST_CONDITION;
        F_EQ_TIME : F_EQ(IN2 := %timeValue%);
        STRINGType : TEST_CONDITION;
        F_EQ_TOD : F_EQ(IN2 := %timeofdayValue%);
        F_EQ_Bool_STRING : F_EQ(IN2 := %stringValue%);
        F_EQ_Bool_WSTRING : F_EQ(IN2 := %wstringValue%);
        TIMEType : TEST_CONDITION;
      END_FBS
      EVENT_CONNECTIONS
        F_EQ_Bool.CNF TO BollType.REQ;
        F_EQ_SINT.CNF TO SINTType.REQ;
        F_EQ_INT.CNF TO INTType.REQ;
        F_EQ_DINT.CNF TO DINType.REQ;
        F_EQ_UINT.CNF TO UINTType.REQ;
        F_EQ_UDINT.CNF TO UDINTType.REQ;
        F_EQ_USINT.CNF TO USINTType.REQ;
        F_EQ_LINT.CNF TO LINTType.REQ;
        F_EQ_WORD.CNF TO WORDType.REQ;
        F_EQ_DWORD.CNF TO DWORDType.REQ;
        F_EQ_BYTE.CNF TO BYTEType.REQ;
        F_EQ_ULINT.CNF TO ULINTType.REQ;
        F_EQ_REAL.CNF TO REALType.REQ;
        F_EQ_TOD.CNF TO TODType.REQ;
        F_EQ_Bool_STRING.CNF TO STRINGType.REQ;
        F_EQ_LREAL.CNF TO LREALType.REQ;
        F_EQ_DT.CNF TO DTType.REQ;
        F_EQ_Bool_WSTRING.CNF TO WSTRINGType.REQ;
        F_EQ_LWORD.CNF TO LWORDType.REQ;
        F_EQ_DATE.CNF TO DATEType.REQ;
        F_EQ_TIME.CNF TO TIMEType.REQ;
        REQ TO F_EQ_Bool.REQ;
        BollType.CNF TO F_EQ_SINT.REQ;
        SINTType.CNF TO F_EQ_INT.REQ;
        INTType.CNF TO F_EQ_DINT.REQ;
        DINType.CNF TO F_EQ_LINT.REQ;
        LINTType.CNF TO F_EQ_USINT.REQ;
        USINTType.CNF TO F_EQ_UINT.REQ;
        UINTType.CNF TO F_EQ_UDINT.REQ;
        UDINTType.CNF TO F_EQ_ULINT.REQ;
        ULINTType.CNF TO F_EQ_BYTE.REQ;
        BYTEType.CNF TO F_EQ_WORD.REQ;
        WORDType.CNF TO F_EQ_DWORD.REQ;
        DWORDType.CNF TO F_EQ_LWORD.REQ;
        DATEType.CNF TO F_EQ_TOD.REQ;
        TODType.CNF TO F_EQ_DT.REQ;
        DTType.CNF TO F_EQ_TIME.REQ;
        TIMEType.CNF TO F_EQ_REAL.REQ;
        REALType.CNF TO F_EQ_LREAL.REQ;
        LREALType.CNF TO F_EQ_Bool_STRING.REQ;
        STRINGType.CNF TO F_EQ_Bool_WSTRING.REQ;
        LWORDType.CNF TO F_EQ_REAL.REQ;
        WSTRINGType.CNF TO CNF;
      END_CONNECTIONS
      DATA_CONNECTIONS
        F_EQ_Bool.OUT TO BollType.check;
        F_EQ_SINT.OUT TO SINTType.check;
        F_EQ_INT.OUT TO INTType.check;
        F_EQ_DINT.OUT TO DINType.check;
        F_EQ_UINT.OUT TO UINTType.check;
        F_EQ_LINT.OUT TO LINTType.check;
        F_EQ_USINT.OUT TO USINTType.check;
        F_EQ_UDINT.OUT TO UDINTType.check;
        F_EQ_WORD.OUT TO WORDType.check;
        F_EQ_ULINT.OUT TO ULINTType.check;
        F_EQ_BYTE.OUT TO BYTEType.check;
        F_EQ_DWORD.OUT TO DWORDType.check;
        F_EQ_TOD.OUT TO TODType.check;
        F_EQ_LWORD.OUT TO LWORDType.check;
        F_EQ_Bool_WSTRING.OUT TO WSTRINGType.check;
        F_EQ_LREAL.OUT TO LREALType.check;
        F_EQ_DATE.OUT TO DATEType.check;
        F_EQ_Bool_STRING.OUT TO STRINGType.check;
        F_EQ_TIME.OUT TO TIMEType.check;
        F_EQ_REAL.OUT TO REALType.check;
        F_EQ_DT.OUT TO DTType.check;
        SINT_I TO F_EQ_SINT.IN1;
        INT_I TO F_EQ_INT.IN1;
        DINT_I TO F_EQ_DINT.IN1;
        LINT_I TO F_EQ_LINT.IN1;
        USINT_I TO F_EQ_USINT.IN1;
        UINT_I TO F_EQ_UINT.IN1;
        UDINT_I TO F_EQ_UDINT.IN1;
        ULINT_I TO F_EQ_ULINT.IN1;
        BYTE_I TO F_EQ_BYTE.IN1;
        WORD_I TO F_EQ_WORD.IN1;
        DWORD_I TO F_EQ_DWORD.IN1;
        LWORD_I TO F_EQ_LWORD.IN1;
        DATE_I TO F_EQ_DATE.IN1;
        TIME_OF_DAY_I TO F_EQ_TOD.IN1;
        DATE_AND_TIME_I TO F_EQ_DT.IN1;
        TIME_I TO F_EQ_TIME.IN1;
        REAL_I TO F_EQ_REAL.IN1;
        LREAL_I TO F_EQ_LREAL.IN1;
        STRING_I TO F_EQ_Bool_STRING.IN1;
        WSTRING_I TO F_EQ_Bool_WSTRING.IN1;
        BOOL_I TO F_EQ_Bool.IN1;
      END_CONNECTIONS
    END_SUBAPPLICATION
    SUBAPPLICATION AllTypes_1
      EVENT_INPUT
        REQ;
      END_EVENT
      EVENT_OUTPUT
        CNF;
      END_EVENT
      VAR_INPUT
        BOOL_I : BOOL; (* BOOL Type Input *)
        SINT_I : SINT; (* SINT Type Input *)
        INT_I : INT; (* INT Type Input *)
        DINT_I : DINT; (* DINT Type Input *)
        LINT_I : LINT; (* LINT Type Input *)
        USINT_I : USINT; (* USINT Type Input *)
        UINT_I : UINT; (* UINT Type Input *)
        UDINT_I : UDINT; (* UDINT Type Input *)
        ULINT_I : ULINT; (* ULINT Type Input *)
        BYTE_I : BYTE; (* BYTE Type Input *)
        WORD_I : WORD; (* WORD Type Input *)
        DWORD_I : DWORD; (* DWORD Type Input *)
        LWORD_I : LWORD; (* LWORD Type Input *)
        DATE_I_BOOL : BOOL; (* DATE Type Input *)
        TIME_OF_DAY_I_BOOL : BOOL; (* TIME_OF_DAY Type Input *)
        DATE_AND_TIME_I_BOOL : BOOL; (* DATE_AND_TIME Type Input *)
        TIME_I : TIME; (* TIME Type Input *)
        REAL_I : REAL; (* REAL Type Input *)
        LREAL_I : LREAL; (* LREAL Type Input *)
        STRING_I : STRING; (* STRING Type Input *)
        WSTRING_I : WSTRING; (* WSTRING Type Input *)
      END_VAR
      VAR_OUTPUT
        BOOL_O : BOOL; (* BOOL Type Output *)
        SINT_O : SINT; (* SINT Type Output *)
        INT_O : INT; (* INT Type Output *)
        DINT_O : DINT; (* DINT Type Output *)
        LINT_O : LINT; (* LINT Type Output *)
        USINT_O : USINT; (* USINT Type Output *)
        UINT_O : UINT; (* UINT Type Output *)
        UDINT_O : UDINT; (* UDINT Type Output *)
        ULINT_O : ULINT; (* ULINT Type Output *)
        BYTE_O : BYTE; (* BYTE Type Output *)
        WORD_O : WORD; (* WORD Type Output *)
        DWORD_O : DWORD; (* DWORD Type Output *)
        LWORD_O : LWORD; (* LWORD Type Output *)
        DATE_O_BOOL : BOOL; (* DATE Type Output *)
        TIME_OF_DAY_O_BOOL : BOOL; (* TIME_OF_DAY Type Output *)
        DATE_AND_TIME_O_BOOL : BOOL; (* DATE_AND_TIME Type Output *)
        TIME_O : TIME; (* TIME Type Output *)
        REAL_O : REAL; (* REAL Type Output *)
        LREAL_O : LREAL; (* LREAL Type Output *)
        STRING_O : STRING; (* STRING Type Output *)
        WSTRING_O : WSTRING; (* WSTRING Type Output *)
      END_VAR
      FBS
        SINT2SINT : SINT2SINT;
        UINT2UINT : UINT2UINT;
        BOOL2BOOL : BOOL2BOOL;
        UDINT2UDINT : UDINT2UDINT;
        DINT2DINT : DINT2DINT;
        F_LINT_TO_INT : F_LINT_TO_INT;
        INT2INT : INT2INT;
        USINT2USINT : USINT2USINT;
        F_ULINT_TO_INT : F_ULINT_TO_INT;
        BYTE2BYTE : BYTE2BYTE;
        WORD2WORD : WORD2WORD;
        DWORD2DWORD : DWORD2DWORD;
        F_LWORD_TO_INT : F_LWORD_TO_INT;
        MISSING_DATE : F_DT_TO_DATE;
        MISSING_DATE_AND_TIME : F_DT_TO_TOD;
        TIME2TIME : TIME2TIME;
        REAL2REAL : REAL2REAL;
        LREAL2LREAL : LREAL2LREAL;
        STRING2STRING : STRING2STRING;
        WSTRING2WSTRING : WSTRING2WSTRING;
        Time_of_day : F_ADD_TOD_TIME;
        F_INT_TO_LINT : F_INT_TO_LINT;
        F_INT_TO_ULINT : F_INT_TO_ULINT;
        F_INT_TO_LWORD : F_INT_TO_LWORD;
        BOOL2BOOL_1 : BOOL2BOOL;
        BOOL2BOOL_2 : BOOL2BOOL;
        BOOL2BOOL_3 : BOOL2BOOL;
      END_FBS
      EVENT_CONNECTIONS
        REQ TO BOOL2BOOL.REQ;
        F_LINT_TO_INT.CNF TO F_INT_TO_LINT.REQ;
        F_ULINT_TO_INT.CNF TO F_INT_TO_ULINT.REQ;
        F_LWORD_TO_INT.CNF TO F_INT_TO_LWORD.REQ;
        BOOL2BOOL.CNF TO SINT2SINT.REQ;
        SINT2SINT.CNF TO INT2INT.REQ;
        INT2INT.CNF TO DINT2DINT.REQ;
        DINT2DINT.CNF TO F_LINT_TO_INT.REQ;
        F_INT_TO_LINT.CNF TO USINT2USINT.REQ;
        USINT2USINT.CNF TO UINT2UINT.REQ;
        UINT2UINT.CNF TO UDINT2UDINT.REQ;
        UDINT2UDINT.CNF TO F_ULINT_TO_INT.REQ;
        F_INT_TO_ULINT.CNF TO BYTE2BYTE.REQ;
        BYTE2BYTE.CNF TO WORD2WORD.REQ;
        WORD2WORD.CNF TO DWORD2DWORD.REQ;
        DWORD2DWORD.CNF TO F_LWORD_TO_INT.REQ;
        F_INT_TO_LWORD.CNF TO BOOL2BOOL_1.REQ;
        BOOL2BOOL_1.CNF TO BOOL2BOOL_2.REQ;
        BOOL2BOOL_2.CNF TO BOOL2BOOL_3.REQ;
        BOOL2BOOL_3.CNF TO TIME2TIME.REQ;
        TIME2TIME.CNF TO REAL2REAL.REQ;
        REAL2REAL.CNF TO LREAL2LREAL.REQ;
        LREAL2LREAL.CNF TO STRING2STRING.REQ;
        STRING2STRING.CNF TO WSTRING2WSTRING.REQ;
        WSTRING2WSTRING.CNF TO CNF;
      END_CONNECTIONS
      DATA_CONNECTIONS
        BOOL_I TO BOOL2BOOL.IN;
        SINT_I TO SINT2SINT.IN;
        INT_I TO INT2INT.IN;
        DINT_I TO DINT2DINT.IN;
        LINT_I TO F_LINT_TO_INT.IN;
        USINT_I TO USINT2USINT.IN;
        UINT_I TO UINT2UINT.IN;
        UDINT_I TO UDINT2UDINT.IN;
        ULINT_I TO F_ULINT_TO_INT.IN;
        BYTE_I TO BYTE2BYTE.IN;
        WORD_I TO WORD2WORD.IN;
        DWORD_I TO DWORD2DWORD.IN;
        LWORD_I TO F_LWORD_TO_INT.IN;
        TIME_I TO TIME2TIME.IN;
        REAL_I TO REAL2REAL.IN;
        LREAL_I TO LREAL2LREAL.IN;
        STRING_I TO STRING2STRING.IN;
        WSTRING_I TO WSTRING2WSTRING.IN;
        SINT2SINT.OUT TO SINT_O;
        INT2INT.OUT TO INT_O;
        DINT2DINT.OUT TO DINT_O;
        F_LINT_TO_INT.OUT TO F_INT_TO_LINT.IN;
        F_INT_TO_LINT.OUT TO LINT_O;
        USINT2USINT.OUT TO USINT_O;
        UINT2UINT.OUT TO UINT_O;
        UDINT2UDINT.OUT TO UDINT_O;
        F_ULINT_TO_INT.OUT TO F_INT_TO_ULINT.IN;
        F_INT_TO_ULINT.OUT TO ULINT_O;
        BYTE2BYTE.OUT TO BYTE_O;
        WORD2WORD.OUT TO WORD_O;
        DWORD2DWORD.OUT TO DWORD_O;
        F_LWORD_TO_INT.OUT TO F_INT_TO_LWORD.IN;
        F_INT_TO_LWORD.OUT TO LWORD_O;
        WSTRING2WSTRING.OUT TO WSTRING_O;
        STRING2STRING.OUT TO STRING_O;
        LREAL2LREAL.OUT TO LREAL_O;
        REAL2REAL.OUT TO REAL_O;
        TIME2TIME.OUT TO TIME_O;
        DATE_I_BOOL TO BOOL2BOOL_1.IN;
        TIME_OF_DAY_I_BOOL TO BOOL2BOOL_2.IN;
        DATE_AND_TIME_I_BOOL TO BOOL2BOOL_3.IN;
        BOOL2BOOL_1.OUT TO DATE_O_BOOL;
        BOOL2BOOL_2.OUT TO TIME_OF_DAY_O_BOOL;
        BOOL2BOOL_3.OUT TO DATE_AND_TIME_O_BOOL;
        BOOL2BOOL.OUT TO BOOL_O;
      END_CONNECTIONS
    END_SUBAPPLICATION
    SUBAPPLICATION HandleInitLocal
      EVENT_INPUT
        InitFinished;
      END_EVENT
      VAR_INPUT
        QI : BOOL;
      END_VAR
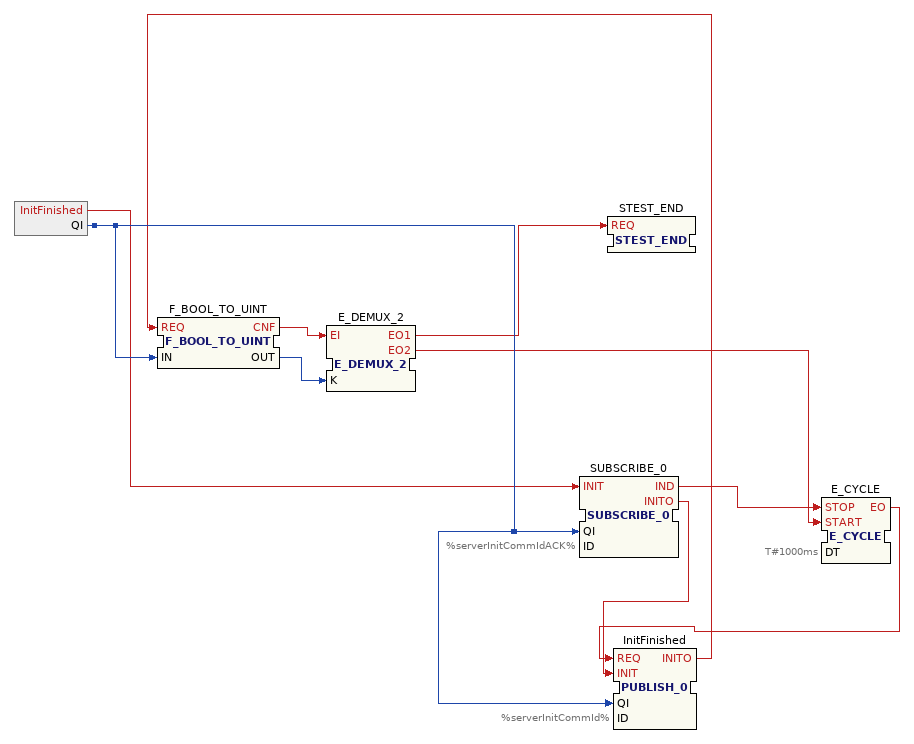
      FBS
        InitFinished : PUBLISH_0(ID := %serverInitCommId%);
        SUBSCRIBE_0 : SUBSCRIBE_0(ID := %serverInitCommIdACK%);
        E_CYCLE : E_CYCLE(DT := T#1000ms);
        E_DEMUX_2 : E_DEMUX_2;
        STEST_END : STEST_END;
        F_BOOL_TO_UINT : F_BOOL_TO_UINT;
      END_FBS
      EVENT_CONNECTIONS
        E_CYCLE.EO TO InitFinished.REQ;
        SUBSCRIBE_0.IND TO E_CYCLE.STOP;
        F_BOOL_TO_UINT.CNF TO E_DEMUX_2.EI;
        E_DEMUX_2.EO1 TO STEST_END.REQ;
        InitFinished TO SUBSCRIBE_0.INIT;
        SUBSCRIBE_0.INITO TO InitFinished.INIT;
        InitFinished.INITO TO F_BOOL_TO_UINT.REQ;
        E_DEMUX_2.EO2 TO E_CYCLE.START;
      END_CONNECTIONS
      DATA_CONNECTIONS
        F_BOOL_TO_UINT.OUT TO E_DEMUX_2.K;
        QI TO F_BOOL_TO_UINT.IN;
        QI TO SUBSCRIBE_0.QI;
        QI TO InitFinished.QI;
      END_CONNECTIONS
    END_SUBAPPLICATION
    SUBAPPLICATION HandleInit
      EVENT_INPUT
        InitFinished;
      END_EVENT
      EVENT_OUTPUT
        Execute;
      END_EVENT
      VAR_INPUT
        QI : BOOL;
      END_VAR
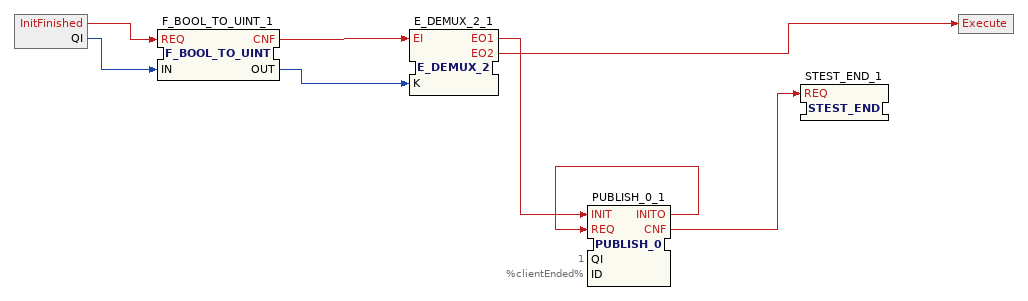
      FBS
        STEST_END_1 : STEST_END;
        E_DEMUX_2_1 : E_DEMUX_2;
        F_BOOL_TO_UINT_1 : F_BOOL_TO_UINT;
        PUBLISH_0_1 : PUBLISH_0(QI := 1, ID := %clientEnded%);
      END_FBS
      EVENT_CONNECTIONS
        F_BOOL_TO_UINT_1.CNF TO E_DEMUX_2_1.EI;
        E_DEMUX_2_1.EO1 TO PUBLISH_0_1.INIT;
        PUBLISH_0_1.INITO TO PUBLISH_0_1.REQ;
        E_DEMUX_2_1.EO2 TO Execute;
        InitFinished TO F_BOOL_TO_UINT_1.REQ;
        PUBLISH_0_1.CNF TO STEST_END_1.REQ;
      END_CONNECTIONS
      DATA_CONNECTIONS
        F_BOOL_TO_UINT_1.OUT TO E_DEMUX_2_1.K;
        QI TO F_BOOL_TO_UINT_1.IN;
      END_CONNECTIONS
    END_SUBAPPLICATION
    SUBAPPLICATION SubApp
      EVENT_INPUT
        REQ;
      END_EVENT
      EVENT_OUTPUT
        CNF;
      END_EVENT
      VAR_OUTPUT
        BOOL_O : BOOL;
        SINT_O : SINT;
        INT_O : INT;
        DINT_O : DINT;
        LINT_O : LINT;
        USINT_O : USINT;
        UINT_O : UINT;
        UDINT_O : UDINT;
        ULINT_O : ULINT;
        BYTE_O : BYTE;
        WORD_o : WORD;
        DWORD_O : DWORD;
        LWORD_O : LWORD;
        DATE_O : BOOL;
        DATE_TIME_O : BOOL;
        TIME_OF_DAY_O : BOOL;
        TIME_O : TIME;
        REAL_O : REAL;
        LREAL_O : LREAL;
        STRING_O : STRING;
        WSTRING_O : WSTRING;
      END_VAR
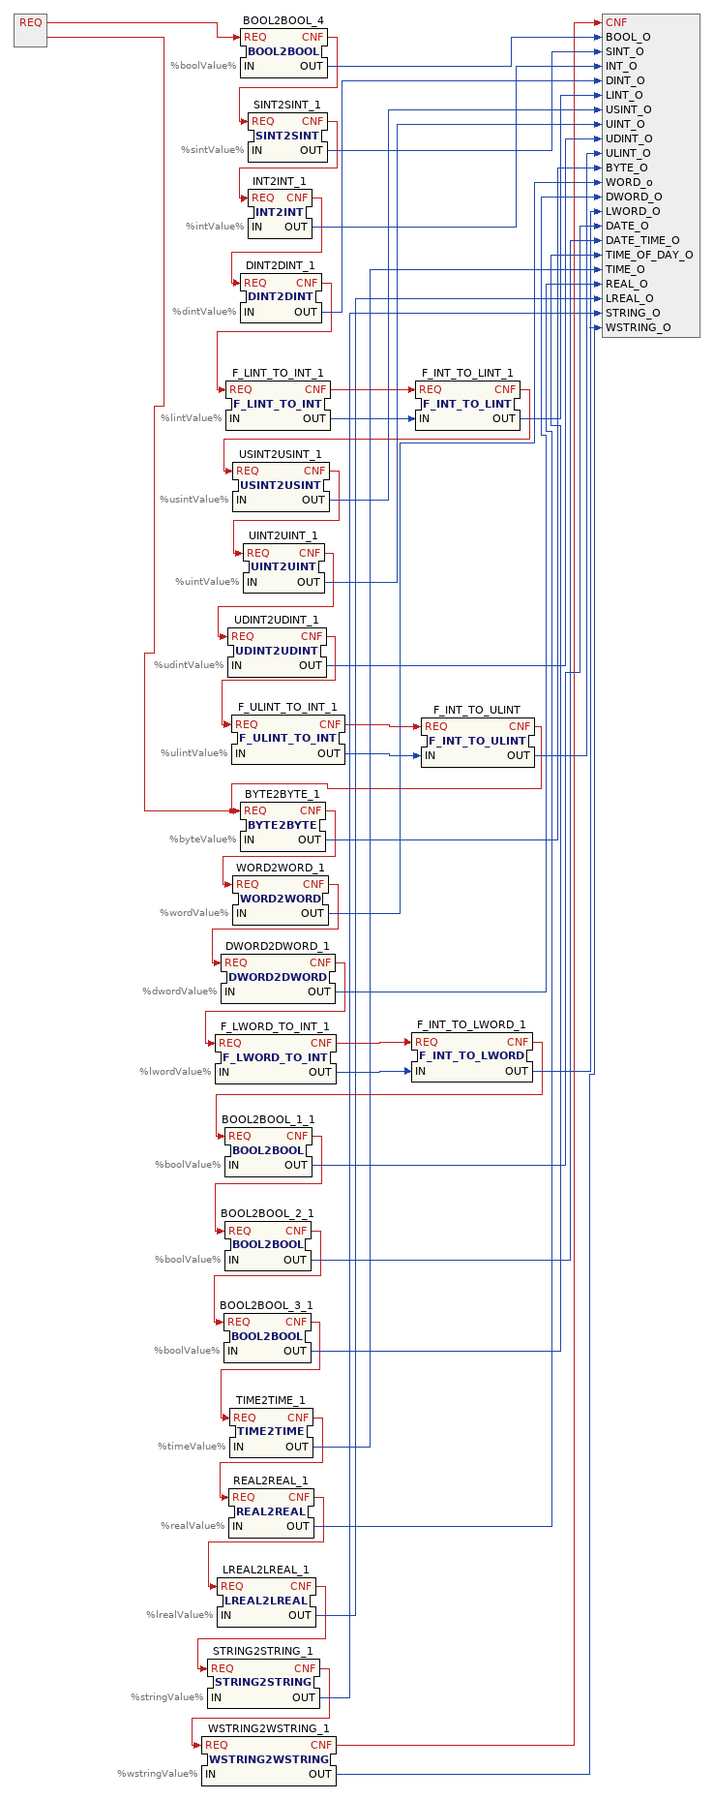
      FBS
        INT2INT_1 : INT2INT(IN := %intValue%);
        BOOL2BOOL_2_1 : BOOL2BOOL(IN := %boolValue%);
        UDINT2UDINT_1 : UDINT2UDINT(IN := %udintValue%);
        SINT2SINT_1 : SINT2SINT(IN := %sintValue%);
        F_INT_TO_LWORD_1 : F_INT_TO_LWORD;
        F_INT_TO_LINT_1 : F_INT_TO_LINT;
        REAL2REAL_1 : REAL2REAL(IN := %realValue%);
        WSTRING2WSTRING_1 : WSTRING2WSTRING(IN := %wstringValue%);
        BYTE2BYTE_1 : BYTE2BYTE(IN := %byteValue%);
        BOOL2BOOL_4 : BOOL2BOOL(IN := %boolValue%);
        BOOL2BOOL_1_1 : BOOL2BOOL(IN := %boolValue%);
        BOOL2BOOL_3_1 : BOOL2BOOL(IN := %boolValue%);
        F_LINT_TO_INT_1 : F_LINT_TO_INT(IN := %lintValue%);
        UINT2UINT_1 : UINT2UINT(IN := %uintValue%);
        STRING2STRING_1 : STRING2STRING(IN := %stringValue%);
        F_ULINT_TO_INT_1 : F_ULINT_TO_INT(IN := %ulintValue%);
        DINT2DINT_1 : DINT2DINT(IN := %dintValue%);
        LREAL2LREAL_1 : LREAL2LREAL(IN := %lrealValue%);
        WORD2WORD_1 : WORD2WORD(IN := %wordValue%);
        F_LWORD_TO_INT_1 : F_LWORD_TO_INT(IN := %lwordValue%);
        USINT2USINT_1 : USINT2USINT(IN := %usintValue%);
        TIME2TIME_1 : TIME2TIME(IN := %timeValue%);
        DWORD2DWORD_1 : DWORD2DWORD(IN := %dwordValue%);
        F_INT_TO_ULINT : F_INT_TO_ULINT;
      END_FBS
      EVENT_CONNECTIONS
        SINT2SINT_1.CNF TO INT2INT_1.REQ;
        INT2INT_1.CNF TO DINT2DINT_1.REQ;
        BOOL2BOOL_1_1.CNF TO BOOL2BOOL_2_1.REQ;
        BOOL2BOOL_2_1.CNF TO BOOL2BOOL_3_1.REQ;
        UINT2UINT_1.CNF TO UDINT2UDINT_1.REQ;
        UDINT2UDINT_1.CNF TO F_ULINT_TO_INT_1.REQ;
        BOOL2BOOL_4.CNF TO SINT2SINT_1.REQ;
        F_LWORD_TO_INT_1.CNF TO F_INT_TO_LWORD_1.REQ;
        F_INT_TO_LWORD_1.CNF TO BOOL2BOOL_1_1.REQ;
        F_LINT_TO_INT_1.CNF TO F_INT_TO_LINT_1.REQ;
        F_INT_TO_LINT_1.CNF TO USINT2USINT_1.REQ;
        TIME2TIME_1.CNF TO REAL2REAL_1.REQ;
        REAL2REAL_1.CNF TO LREAL2LREAL_1.REQ;
        STRING2STRING_1.CNF TO WSTRING2WSTRING_1.REQ;
         TO BYTE2BYTE_1.REQ;
        BYTE2BYTE_1.CNF TO WORD2WORD_1.REQ;
        BOOL2BOOL_3_1.CNF TO TIME2TIME_1.REQ;
        DINT2DINT_1.CNF TO F_LINT_TO_INT_1.REQ;
        USINT2USINT_1.CNF TO UINT2UINT_1.REQ;
        LREAL2LREAL_1.CNF TO STRING2STRING_1.REQ;
        WORD2WORD_1.CNF TO DWORD2DWORD_1.REQ;
        DWORD2DWORD_1.CNF TO F_LWORD_TO_INT_1.REQ;
        WSTRING2WSTRING_1.CNF TO CNF;
        REQ TO BOOL2BOOL_4.REQ;
        F_ULINT_TO_INT_1.CNF TO F_INT_TO_ULINT.REQ;
        F_INT_TO_ULINT.CNF TO BYTE2BYTE_1.REQ;
      END_CONNECTIONS
      DATA_CONNECTIONS
        F_LWORD_TO_INT_1.OUT TO F_INT_TO_LWORD_1.IN;
        F_LINT_TO_INT_1.OUT TO F_INT_TO_LINT_1.IN;
        INT2INT_1.OUT TO INT_O;
        BOOL2BOOL_2_1.OUT TO DATE_TIME_O;
        UDINT2UDINT_1.OUT TO UDINT_O;
        SINT2SINT_1.OUT TO SINT_O;
        F_INT_TO_LWORD_1.OUT TO LWORD_O;
        F_INT_TO_LINT_1.OUT TO LINT_O;
        REAL2REAL_1.OUT TO REAL_O;
        WSTRING2WSTRING_1.OUT TO WSTRING_O;
        BYTE2BYTE_1.OUT TO BYTE_O;
        BOOL2BOOL_4.OUT TO BOOL_O;
        BOOL2BOOL_1_1.OUT TO DATE_O;
        BOOL2BOOL_3_1.OUT TO TIME_OF_DAY_O;
        UINT2UINT_1.OUT TO UINT_O;
        STRING2STRING_1.OUT TO STRING_O;
        DINT2DINT_1.OUT TO DINT_O;
        LREAL2LREAL_1.OUT TO LREAL_O;
        WORD2WORD_1.OUT TO WORD_o;
        USINT2USINT_1.OUT TO USINT_O;
        TIME2TIME_1.OUT TO TIME_O;
        DWORD2DWORD_1.OUT TO DWORD_O;
        F_INT_TO_ULINT.OUT TO ULINT_O;
        F_ULINT_TO_INT_1.OUT TO F_INT_TO_ULINT.IN;
      END_CONNECTIONS
    END_SUBAPPLICATION
    SUBAPPLICATION TypeTest_2
      EVENT_INPUT
        REQ;
      END_EVENT
      EVENT_OUTPUT
        CNF;
      END_EVENT
      VAR_INPUT
        BOOL_I : BOOL; (* BOOL Type Input *)
        SINT_I : SINT; (* SINT Type Input *)
        INT_I : INT; (* INT Type Input *)
        DINT_I : DINT; (* DINT Type Input *)
        LINT_I : LINT; (* LINT Type Input *)
        USINT_I : USINT; (* USINT Type Input *)
        UINT_I : UINT; (* UINT Type Input *)
        UDINT_I : UDINT; (* UDINT Type Input *)
        ULINT_I : ULINT; (* ULINT Type Input *)
        BYTE_I : BYTE; (* BYTE Type Input *)
        WORD_I : WORD; (* WORD Type Input *)
        DWORD_I : DWORD; (* DWORD Type Input *)
        LWORD_I : LWORD; (* LWORD Type Input *)
        DATE_I : DATE; (* DATE Type Input *)
        TIME_OF_DAY_I : TIME_OF_DAY; (* TIME_OF_DAY Type Input *)
        DATE_AND_TIME_I : DATE_AND_TIME; (* DATE_AND_TIME Type Input *)
        TIME_I : TIME; (* TIME Type Input *)
        REAL_I : REAL; (* REAL Type Input *)
        LREAL_I : LREAL; (* LREAL Type Input *)
        STRING_I : STRING; (* STRING Type Input *)
        WSTRING_I : WSTRING; (* WSTRING Type Input *)
      END_VAR
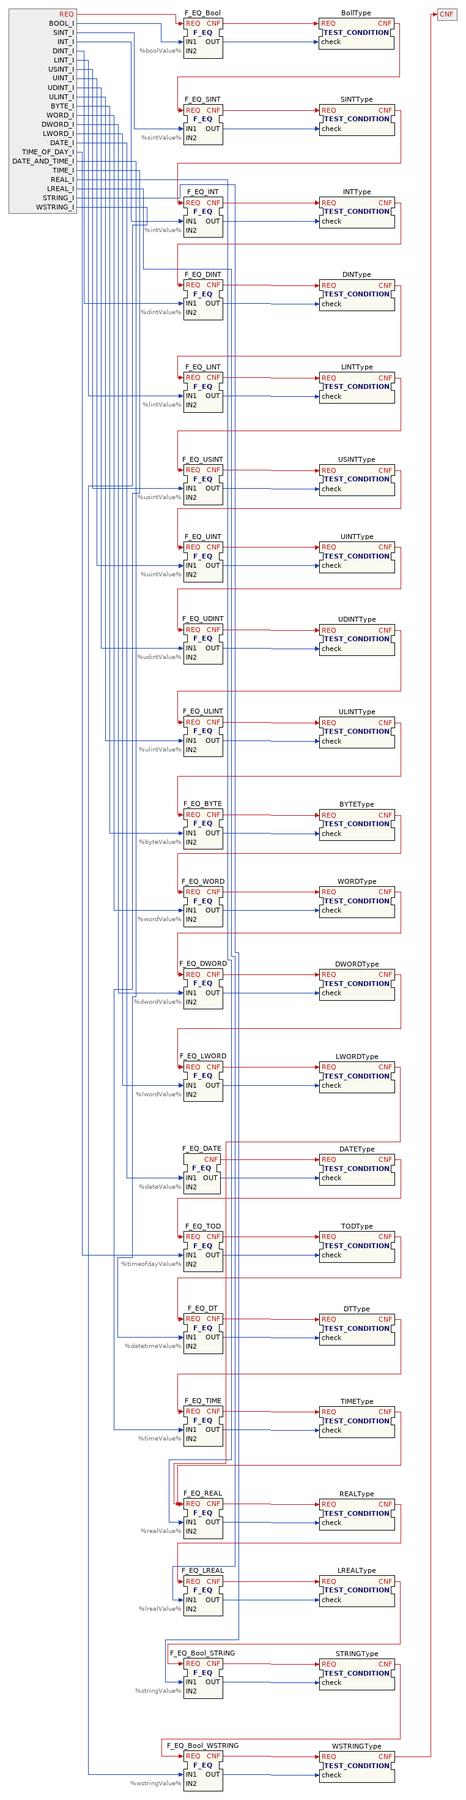
      FBS
        BollType : TEST_CONDITION;
        F_EQ_Bool : F_EQ(IN2 := %boolValue%);
        SINTType : TEST_CONDITION;
        F_EQ_SINT : F_EQ(IN2 := %sintValue%);
        INTType : TEST_CONDITION;
        F_EQ_INT : F_EQ(IN2 := %intValue%);
        DINType : TEST_CONDITION;
        F_EQ_DINT : F_EQ(IN2 := %dintValue%);
        F_EQ_USINT : F_EQ(IN2 := %usintValue%);
        USINTType : TEST_CONDITION;
        F_EQ_UINT : F_EQ(IN2 := %uintValue%);
        LINTType : TEST_CONDITION;
        UINTType : TEST_CONDITION;
        UDINTType : TEST_CONDITION;
        F_EQ_UDINT : F_EQ(IN2 := %udintValue%);
        F_EQ_LINT : F_EQ(IN2 := %lintValue%);
        F_EQ_BYTE : F_EQ(IN2 := %byteValue%);
        BYTEType : TEST_CONDITION;
        F_EQ_WORD : F_EQ(IN2 := %wordValue%);
        ULINTType : TEST_CONDITION;
        WORDType : TEST_CONDITION;
        DWORDType : TEST_CONDITION;
        F_EQ_DWORD : F_EQ(IN2 := %dwordValue%);
        F_EQ_ULINT : F_EQ(IN2 := %ulintValue%);
        F_EQ_DATE : F_EQ(IN2 := %dateValue%);
        DATEType : TEST_CONDITION;
        F_EQ_LREAL : F_EQ(IN2 := %lrealValue%);
        LWORDType : TEST_CONDITION;
        TODType : TEST_CONDITION;
        DTType : TEST_CONDITION;
        F_EQ_DT : F_EQ(IN2 := %datetimeValue%);
        REALType : TEST_CONDITION;
        LREALType : TEST_CONDITION;
        F_EQ_REAL : F_EQ(IN2 := %realValue%);
        F_EQ_LWORD : F_EQ(IN2 := %lwordValue%);
        WSTRINGType : TEST_CONDITION;
        F_EQ_TIME : F_EQ(IN2 := %timeValue%);
        STRINGType : TEST_CONDITION;
        F_EQ_TOD : F_EQ(IN2 := %timeofdayValue%);
        F_EQ_Bool_STRING : F_EQ(IN2 := %stringValue%);
        F_EQ_Bool_WSTRING : F_EQ(IN2 := %wstringValue%);
        TIMEType : TEST_CONDITION;
      END_FBS
      EVENT_CONNECTIONS
        F_EQ_Bool.CNF TO BollType.REQ;
        F_EQ_SINT.CNF TO SINTType.REQ;
        F_EQ_INT.CNF TO INTType.REQ;
        F_EQ_DINT.CNF TO DINType.REQ;
        F_EQ_UINT.CNF TO UINTType.REQ;
        F_EQ_UDINT.CNF TO UDINTType.REQ;
        F_EQ_USINT.CNF TO USINTType.REQ;
        F_EQ_LINT.CNF TO LINTType.REQ;
        F_EQ_WORD.CNF TO WORDType.REQ;
        F_EQ_DWORD.CNF TO DWORDType.REQ;
        F_EQ_BYTE.CNF TO BYTEType.REQ;
        F_EQ_ULINT.CNF TO ULINTType.REQ;
        F_EQ_REAL.CNF TO REALType.REQ;
        F_EQ_TOD.CNF TO TODType.REQ;
        F_EQ_Bool_STRING.CNF TO STRINGType.REQ;
        F_EQ_LREAL.CNF TO LREALType.REQ;
        F_EQ_DT.CNF TO DTType.REQ;
        F_EQ_Bool_WSTRING.CNF TO WSTRINGType.REQ;
        F_EQ_LWORD.CNF TO LWORDType.REQ;
        F_EQ_DATE.CNF TO DATEType.REQ;
        F_EQ_TIME.CNF TO TIMEType.REQ;
        REQ TO F_EQ_Bool.REQ;
        BollType.CNF TO F_EQ_SINT.REQ;
        SINTType.CNF TO F_EQ_INT.REQ;
        INTType.CNF TO F_EQ_DINT.REQ;
        DINType.CNF TO F_EQ_LINT.REQ;
        LINTType.CNF TO F_EQ_USINT.REQ;
        USINTType.CNF TO F_EQ_UINT.REQ;
        UINTType.CNF TO F_EQ_UDINT.REQ;
        UDINTType.CNF TO F_EQ_ULINT.REQ;
        ULINTType.CNF TO F_EQ_BYTE.REQ;
        BYTEType.CNF TO F_EQ_WORD.REQ;
        WORDType.CNF TO F_EQ_DWORD.REQ;
        DWORDType.CNF TO F_EQ_LWORD.REQ;
        DATEType.CNF TO F_EQ_TOD.REQ;
        TODType.CNF TO F_EQ_DT.REQ;
        DTType.CNF TO F_EQ_TIME.REQ;
        TIMEType.CNF TO F_EQ_REAL.REQ;
        REALType.CNF TO F_EQ_LREAL.REQ;
        LREALType.CNF TO F_EQ_Bool_STRING.REQ;
        STRINGType.CNF TO F_EQ_Bool_WSTRING.REQ;
        LWORDType.CNF TO F_EQ_REAL.REQ;
        WSTRINGType.CNF TO CNF;
      END_CONNECTIONS
      DATA_CONNECTIONS
        F_EQ_Bool.OUT TO BollType.check;
        F_EQ_SINT.OUT TO SINTType.check;
        F_EQ_INT.OUT TO INTType.check;
        F_EQ_DINT.OUT TO DINType.check;
        F_EQ_UINT.OUT TO UINTType.check;
        F_EQ_LINT.OUT TO LINTType.check;
        F_EQ_USINT.OUT TO USINTType.check;
        F_EQ_UDINT.OUT TO UDINTType.check;
        F_EQ_WORD.OUT TO WORDType.check;
        F_EQ_ULINT.OUT TO ULINTType.check;
        F_EQ_BYTE.OUT TO BYTEType.check;
        F_EQ_DWORD.OUT TO DWORDType.check;
        F_EQ_TOD.OUT TO TODType.check;
        F_EQ_LWORD.OUT TO LWORDType.check;
        F_EQ_Bool_WSTRING.OUT TO WSTRINGType.check;
        F_EQ_LREAL.OUT TO LREALType.check;
        F_EQ_DATE.OUT TO DATEType.check;
        F_EQ_Bool_STRING.OUT TO STRINGType.check;
        F_EQ_TIME.OUT TO TIMEType.check;
        F_EQ_REAL.OUT TO REALType.check;
        F_EQ_DT.OUT TO DTType.check;
        SINT_I TO F_EQ_SINT.IN1;
        INT_I TO F_EQ_INT.IN1;
        DINT_I TO F_EQ_DINT.IN1;
        LINT_I TO F_EQ_LINT.IN1;
        USINT_I TO F_EQ_USINT.IN1;
        UINT_I TO F_EQ_UINT.IN1;
        UDINT_I TO F_EQ_UDINT.IN1;
        ULINT_I TO F_EQ_ULINT.IN1;
        BYTE_I TO F_EQ_BYTE.IN1;
        WORD_I TO F_EQ_WORD.IN1;
        DWORD_I TO F_EQ_DWORD.IN1;
        LWORD_I TO F_EQ_LWORD.IN1;
        DATE_I TO F_EQ_DATE.IN1;
        TIME_OF_DAY_I TO F_EQ_TOD.IN1;
        DATE_AND_TIME_I TO F_EQ_DT.IN1;
        TIME_I TO F_EQ_TIME.IN1;
        REAL_I TO F_EQ_REAL.IN1;
        LREAL_I TO F_EQ_LREAL.IN1;
        STRING_I TO F_EQ_Bool_STRING.IN1;
        WSTRING_I TO F_EQ_Bool_WSTRING.IN1;
        BOOL_I TO F_EQ_Bool.IN1;
      END_CONNECTIONS
    END_SUBAPPLICATION
    SUBAPPLICATION SubApp_1
      EVENT_INPUT
        REQ;
      END_EVENT
      EVENT_OUTPUT
        CNF;
      END_EVENT
      VAR_OUTPUT
        BOOL_O : BOOL;
        SINT_O : SINT;
        INT_O : INT;
        DINT_O : DINT;
        LINT_O : LINT;
        USINT_O : USINT;
        UINT_O : UINT;
        UDINT_O : UDINT;
        ULINT_O : ULINT;
        BYTE_O : BYTE;
        WORD_O : WORD;
        DWORD_O : DWORD;
        LWORD_O : LWORD;
        DATE_O : BOOL;
        DATE_TIME_O : BOOL;
        TIME_OF_DAY_O : BOOL;
        TIME_O : TIME;
        REAL_O : REAL;
        LREAL_O : LREAL;
        STRING_O : STRING;
        WSTRING_O : WSTRING;
      END_VAR
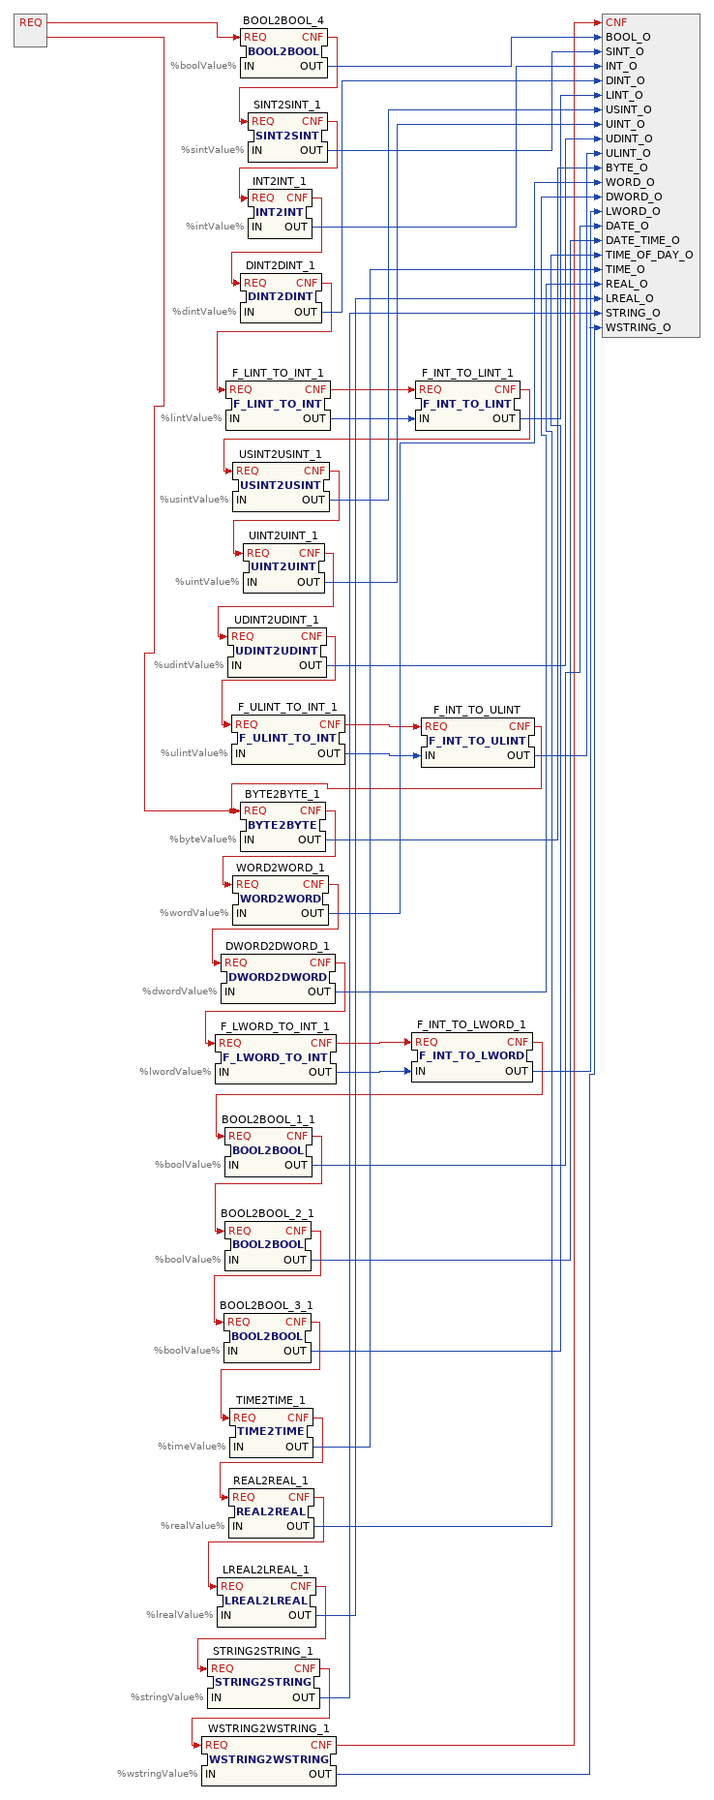
      FBS
        INT2INT_1 : INT2INT(IN := %intValue%);
        BOOL2BOOL_2_1 : BOOL2BOOL(IN := %boolValue%);
        UDINT2UDINT_1 : UDINT2UDINT(IN := %udintValue%);
        SINT2SINT_1 : SINT2SINT(IN := %sintValue%);
        F_INT_TO_LWORD_1 : F_INT_TO_LWORD;
        F_INT_TO_LINT_1 : F_INT_TO_LINT;
        REAL2REAL_1 : REAL2REAL(IN := %realValue%);
        WSTRING2WSTRING_1 : WSTRING2WSTRING(IN := %wstringValue%);
        BYTE2BYTE_1 : BYTE2BYTE(IN := %byteValue%);
        BOOL2BOOL_4 : BOOL2BOOL(IN := %boolValue%);
        BOOL2BOOL_1_1 : BOOL2BOOL(IN := %boolValue%);
        BOOL2BOOL_3_1 : BOOL2BOOL(IN := %boolValue%);
        F_LINT_TO_INT_1 : F_LINT_TO_INT(IN := %lintValue%);
        UINT2UINT_1 : UINT2UINT(IN := %uintValue%);
        STRING2STRING_1 : STRING2STRING(IN := %stringValue%);
        F_ULINT_TO_INT_1 : F_ULINT_TO_INT(IN := %ulintValue%);
        DINT2DINT_1 : DINT2DINT(IN := %dintValue%);
        LREAL2LREAL_1 : LREAL2LREAL(IN := %lrealValue%);
        WORD2WORD_1 : WORD2WORD(IN := %wordValue%);
        F_LWORD_TO_INT_1 : F_LWORD_TO_INT(IN := %lwordValue%);
        USINT2USINT_1 : USINT2USINT(IN := %usintValue%);
        TIME2TIME_1 : TIME2TIME(IN := %timeValue%);
        DWORD2DWORD_1 : DWORD2DWORD(IN := %dwordValue%);
        F_INT_TO_ULINT : F_INT_TO_ULINT;
      END_FBS
      EVENT_CONNECTIONS
        SINT2SINT_1.CNF TO INT2INT_1.REQ;
        INT2INT_1.CNF TO DINT2DINT_1.REQ;
        BOOL2BOOL_1_1.CNF TO BOOL2BOOL_2_1.REQ;
        BOOL2BOOL_2_1.CNF TO BOOL2BOOL_3_1.REQ;
        UINT2UINT_1.CNF TO UDINT2UDINT_1.REQ;
        UDINT2UDINT_1.CNF TO F_ULINT_TO_INT_1.REQ;
        BOOL2BOOL_4.CNF TO SINT2SINT_1.REQ;
        F_LWORD_TO_INT_1.CNF TO F_INT_TO_LWORD_1.REQ;
        F_INT_TO_LWORD_1.CNF TO BOOL2BOOL_1_1.REQ;
        F_LINT_TO_INT_1.CNF TO F_INT_TO_LINT_1.REQ;
        F_INT_TO_LINT_1.CNF TO USINT2USINT_1.REQ;
        TIME2TIME_1.CNF TO REAL2REAL_1.REQ;
        REAL2REAL_1.CNF TO LREAL2LREAL_1.REQ;
        STRING2STRING_1.CNF TO WSTRING2WSTRING_1.REQ;
         TO BYTE2BYTE_1.REQ;
        BYTE2BYTE_1.CNF TO WORD2WORD_1.REQ;
        BOOL2BOOL_3_1.CNF TO TIME2TIME_1.REQ;
        DINT2DINT_1.CNF TO F_LINT_TO_INT_1.REQ;
        USINT2USINT_1.CNF TO UINT2UINT_1.REQ;
        LREAL2LREAL_1.CNF TO STRING2STRING_1.REQ;
        WORD2WORD_1.CNF TO DWORD2DWORD_1.REQ;
        DWORD2DWORD_1.CNF TO F_LWORD_TO_INT_1.REQ;
        WSTRING2WSTRING_1.CNF TO CNF;
        REQ TO BOOL2BOOL_4.REQ;
        F_ULINT_TO_INT_1.CNF TO F_INT_TO_ULINT.REQ;
        F_INT_TO_ULINT.CNF TO BYTE2BYTE_1.REQ;
      END_CONNECTIONS
      DATA_CONNECTIONS
        F_LWORD_TO_INT_1.OUT TO F_INT_TO_LWORD_1.IN;
        F_LINT_TO_INT_1.OUT TO F_INT_TO_LINT_1.IN;
        INT2INT_1.OUT TO INT_O;
        BOOL2BOOL_2_1.OUT TO DATE_TIME_O;
        UDINT2UDINT_1.OUT TO UDINT_O;
        SINT2SINT_1.OUT TO SINT_O;
        F_INT_TO_LWORD_1.OUT TO LWORD_O;
        F_INT_TO_LINT_1.OUT TO LINT_O;
        REAL2REAL_1.OUT TO REAL_O;
        WSTRING2WSTRING_1.OUT TO WSTRING_O;
        BYTE2BYTE_1.OUT TO BYTE_O;
        BOOL2BOOL_4.OUT TO BOOL_O;
        BOOL2BOOL_1_1.OUT TO DATE_O;
        BOOL2BOOL_3_1.OUT TO TIME_OF_DAY_O;
        UINT2UINT_1.OUT TO UINT_O;
        STRING2STRING_1.OUT TO STRING_O;
        DINT2DINT_1.OUT TO DINT_O;
        LREAL2LREAL_1.OUT TO LREAL_O;
        WORD2WORD_1.OUT TO WORD_O;
        USINT2USINT_1.OUT TO USINT_O;
        TIME2TIME_1.OUT TO TIME_O;
        DWORD2DWORD_1.OUT TO DWORD_O;
        F_INT_TO_ULINT.OUT TO ULINT_O;
        F_ULINT_TO_INT_1.OUT TO F_INT_TO_ULINT.IN;
      END_CONNECTIONS
    END_SUBAPPLICATION
    SUBAPPLICATION SubApp_2
      EVENT_INPUT
        REQ;
      END_EVENT
      EVENT_OUTPUT
        CNF;
      END_EVENT
      VAR_OUTPUT
        BOOL_O : BOOL;
        SINT_O : SINT;
        INT_O : INT;
        DINT_O : DINT;
        LINT_O : LINT;
        USINT_O : USINT;
        UINT_O : UINT;
        UDINT_O : UDINT;
        ULINT_O : ULINT;
        BYTE_O : BYTE;
        WORD_O : WORD;
        DWORD_O : DWORD;
        LWORD_O : LWORD;
        DATE_O : BOOL;
        DATE_TIME_O : BOOL;
        TIME_OF_DAY_O : BOOL;
        TIME_O : TIME;
        REAL_O : REAL;
        LREAL_O : LREAL;
        STRING_O : STRING;
        WSTRING_O : WSTRING;
      END_VAR
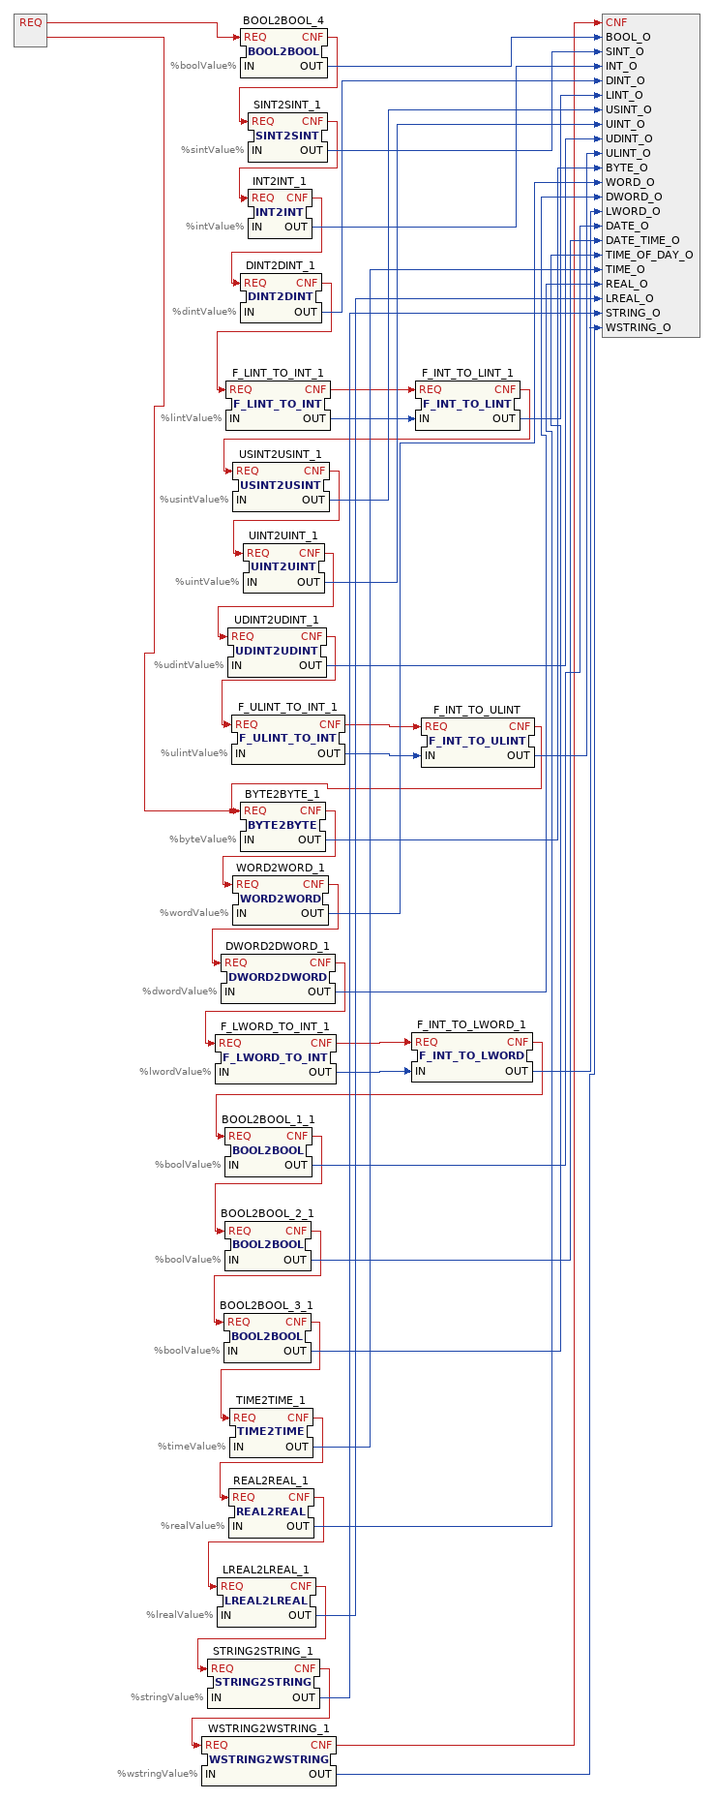
      FBS
        INT2INT_1 : INT2INT(IN := %intValue%);
        BOOL2BOOL_2_1 : BOOL2BOOL(IN := %boolValue%);
        UDINT2UDINT_1 : UDINT2UDINT(IN := %udintValue%);
        SINT2SINT_1 : SINT2SINT(IN := %sintValue%);
        F_INT_TO_LWORD_1 : F_INT_TO_LWORD;
        F_INT_TO_LINT_1 : F_INT_TO_LINT;
        REAL2REAL_1 : REAL2REAL(IN := %realValue%);
        WSTRING2WSTRING_1 : WSTRING2WSTRING(IN := %wstringValue%);
        BYTE2BYTE_1 : BYTE2BYTE(IN := %byteValue%);
        BOOL2BOOL_4 : BOOL2BOOL(IN := %boolValue%);
        BOOL2BOOL_1_1 : BOOL2BOOL(IN := %boolValue%);
        BOOL2BOOL_3_1 : BOOL2BOOL(IN := %boolValue%);
        F_LINT_TO_INT_1 : F_LINT_TO_INT(IN := %lintValue%);
        UINT2UINT_1 : UINT2UINT(IN := %uintValue%);
        STRING2STRING_1 : STRING2STRING(IN := %stringValue%);
        F_ULINT_TO_INT_1 : F_ULINT_TO_INT(IN := %ulintValue%);
        DINT2DINT_1 : DINT2DINT(IN := %dintValue%);
        LREAL2LREAL_1 : LREAL2LREAL(IN := %lrealValue%);
        WORD2WORD_1 : WORD2WORD(IN := %wordValue%);
        F_LWORD_TO_INT_1 : F_LWORD_TO_INT(IN := %lwordValue%);
        USINT2USINT_1 : USINT2USINT(IN := %usintValue%);
        TIME2TIME_1 : TIME2TIME(IN := %timeValue%);
        DWORD2DWORD_1 : DWORD2DWORD(IN := %dwordValue%);
        F_INT_TO_ULINT : F_INT_TO_ULINT;
      END_FBS
      EVENT_CONNECTIONS
        SINT2SINT_1.CNF TO INT2INT_1.REQ;
        INT2INT_1.CNF TO DINT2DINT_1.REQ;
        BOOL2BOOL_1_1.CNF TO BOOL2BOOL_2_1.REQ;
        BOOL2BOOL_2_1.CNF TO BOOL2BOOL_3_1.REQ;
        UINT2UINT_1.CNF TO UDINT2UDINT_1.REQ;
        UDINT2UDINT_1.CNF TO F_ULINT_TO_INT_1.REQ;
        BOOL2BOOL_4.CNF TO SINT2SINT_1.REQ;
        F_LWORD_TO_INT_1.CNF TO F_INT_TO_LWORD_1.REQ;
        F_INT_TO_LWORD_1.CNF TO BOOL2BOOL_1_1.REQ;
        F_LINT_TO_INT_1.CNF TO F_INT_TO_LINT_1.REQ;
        F_INT_TO_LINT_1.CNF TO USINT2USINT_1.REQ;
        TIME2TIME_1.CNF TO REAL2REAL_1.REQ;
        REAL2REAL_1.CNF TO LREAL2LREAL_1.REQ;
        STRING2STRING_1.CNF TO WSTRING2WSTRING_1.REQ;
         TO BYTE2BYTE_1.REQ;
        BYTE2BYTE_1.CNF TO WORD2WORD_1.REQ;
        BOOL2BOOL_3_1.CNF TO TIME2TIME_1.REQ;
        DINT2DINT_1.CNF TO F_LINT_TO_INT_1.REQ;
        USINT2USINT_1.CNF TO UINT2UINT_1.REQ;
        LREAL2LREAL_1.CNF TO STRING2STRING_1.REQ;
        WORD2WORD_1.CNF TO DWORD2DWORD_1.REQ;
        DWORD2DWORD_1.CNF TO F_LWORD_TO_INT_1.REQ;
        WSTRING2WSTRING_1.CNF TO CNF;
        REQ TO BOOL2BOOL_4.REQ;
        F_ULINT_TO_INT_1.CNF TO F_INT_TO_ULINT.REQ;
        F_INT_TO_ULINT.CNF TO BYTE2BYTE_1.REQ;
      END_CONNECTIONS
      DATA_CONNECTIONS
        F_LWORD_TO_INT_1.OUT TO F_INT_TO_LWORD_1.IN;
        F_LINT_TO_INT_1.OUT TO F_INT_TO_LINT_1.IN;
        INT2INT_1.OUT TO INT_O;
        BOOL2BOOL_2_1.OUT TO DATE_TIME_O;
        UDINT2UDINT_1.OUT TO UDINT_O;
        SINT2SINT_1.OUT TO SINT_O;
        F_INT_TO_LWORD_1.OUT TO LWORD_O;
        F_INT_TO_LINT_1.OUT TO LINT_O;
        REAL2REAL_1.OUT TO REAL_O;
        WSTRING2WSTRING_1.OUT TO WSTRING_O;
        BYTE2BYTE_1.OUT TO BYTE_O;
        BOOL2BOOL_4.OUT TO BOOL_O;
        BOOL2BOOL_1_1.OUT TO DATE_O;
        BOOL2BOOL_3_1.OUT TO TIME_OF_DAY_O;
        UINT2UINT_1.OUT TO UINT_O;
        STRING2STRING_1.OUT TO STRING_O;
        DINT2DINT_1.OUT TO DINT_O;
        LREAL2LREAL_1.OUT TO LREAL_O;
        WORD2WORD_1.OUT TO WORD_O;
        USINT2USINT_1.OUT TO USINT_O;
        TIME2TIME_1.OUT TO TIME_O;
        DWORD2DWORD_1.OUT TO DWORD_O;
        F_INT_TO_ULINT.OUT TO ULINT_O;
        F_ULINT_TO_INT_1.OUT TO F_INT_TO_ULINT.IN;
      END_CONNECTIONS
    END_SUBAPPLICATION
    SUBAPPLICATION TypeTest_3
      EVENT_INPUT
        REQ;
      END_EVENT
      EVENT_OUTPUT
        CNF;
      END_EVENT
      VAR_INPUT
        BOOL_I : BOOL; (* BOOL Type Input *)
        SINT_I : SINT; (* SINT Type Input *)
        INT_I : INT; (* INT Type Input *)
        DINT_I : DINT; (* DINT Type Input *)
        LINT_I : LINT; (* LINT Type Input *)
        USINT_I : USINT; (* USINT Type Input *)
        UINT_I : UINT; (* UINT Type Input *)
        UDINT_I : UDINT; (* UDINT Type Input *)
        ULINT_I : ULINT; (* ULINT Type Input *)
        BYTE_I : BYTE; (* BYTE Type Input *)
        WORD_I : WORD; (* WORD Type Input *)
        DWORD_I : DWORD; (* DWORD Type Input *)
        LWORD_I : LWORD; (* LWORD Type Input *)
        DATE_I : DATE; (* DATE Type Input *)
        TIME_OF_DAY_I : TIME_OF_DAY; (* TIME_OF_DAY Type Input *)
        DATE_AND_TIME_I : DATE_AND_TIME; (* DATE_AND_TIME Type Input *)
        TIME_I : TIME; (* TIME Type Input *)
        REAL_I : REAL; (* REAL Type Input *)
        LREAL_I : LREAL; (* LREAL Type Input *)
        STRING_I : STRING; (* STRING Type Input *)
        WSTRING_I : WSTRING; (* WSTRING Type Input *)
      END_VAR
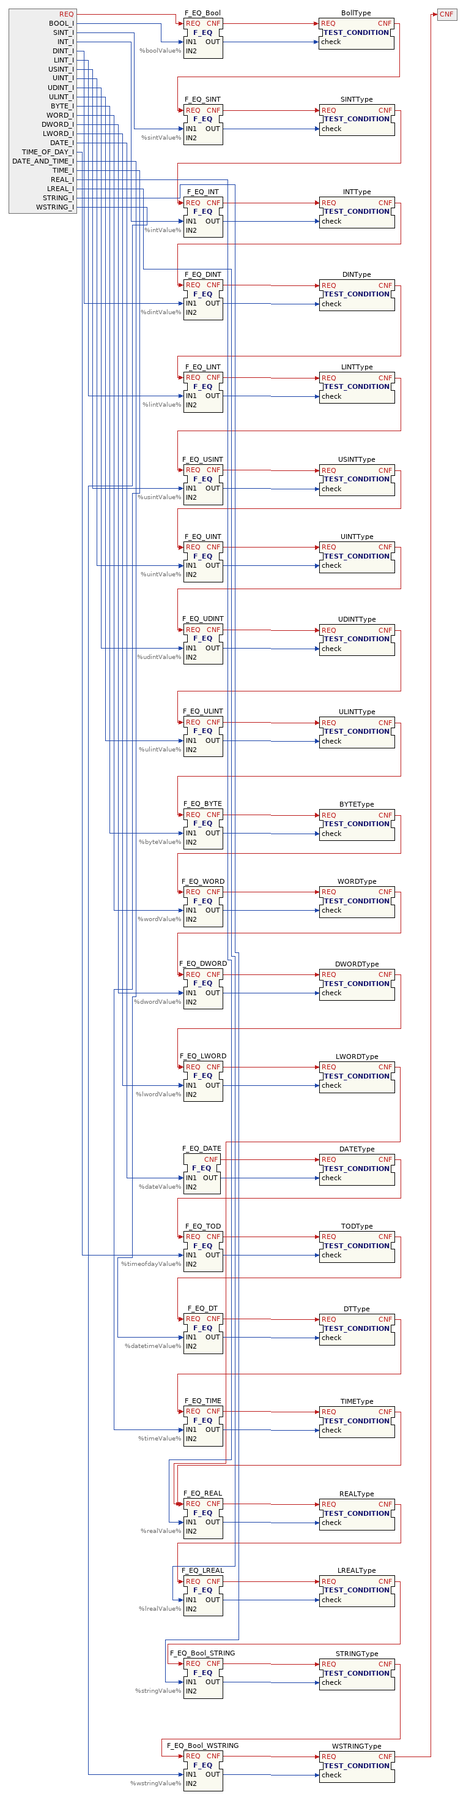
      FBS
        BollType : TEST_CONDITION;
        F_EQ_Bool : F_EQ(IN2 := %boolValue%);
        SINTType : TEST_CONDITION;
        F_EQ_SINT : F_EQ(IN2 := %sintValue%);
        INTType : TEST_CONDITION;
        F_EQ_INT : F_EQ(IN2 := %intValue%);
        DINType : TEST_CONDITION;
        F_EQ_DINT : F_EQ(IN2 := %dintValue%);
        F_EQ_USINT : F_EQ(IN2 := %usintValue%);
        USINTType : TEST_CONDITION;
        F_EQ_UINT : F_EQ(IN2 := %uintValue%);
        LINTType : TEST_CONDITION;
        UINTType : TEST_CONDITION;
        UDINTType : TEST_CONDITION;
        F_EQ_UDINT : F_EQ(IN2 := %udintValue%);
        F_EQ_LINT : F_EQ(IN2 := %lintValue%);
        F_EQ_BYTE : F_EQ(IN2 := %byteValue%);
        BYTEType : TEST_CONDITION;
        F_EQ_WORD : F_EQ(IN2 := %wordValue%);
        ULINTType : TEST_CONDITION;
        WORDType : TEST_CONDITION;
        DWORDType : TEST_CONDITION;
        F_EQ_DWORD : F_EQ(IN2 := %dwordValue%);
        F_EQ_ULINT : F_EQ(IN2 := %ulintValue%);
        F_EQ_DATE : F_EQ(IN2 := %dateValue%);
        DATEType : TEST_CONDITION;
        F_EQ_LREAL : F_EQ(IN2 := %lrealValue%);
        LWORDType : TEST_CONDITION;
        TODType : TEST_CONDITION;
        DTType : TEST_CONDITION;
        F_EQ_DT : F_EQ(IN2 := %datetimeValue%);
        REALType : TEST_CONDITION;
        LREALType : TEST_CONDITION;
        F_EQ_REAL : F_EQ(IN2 := %realValue%);
        F_EQ_LWORD : F_EQ(IN2 := %lwordValue%);
        WSTRINGType : TEST_CONDITION;
        F_EQ_TIME : F_EQ(IN2 := %timeValue%);
        STRINGType : TEST_CONDITION;
        F_EQ_TOD : F_EQ(IN2 := %timeofdayValue%);
        F_EQ_Bool_STRING : F_EQ(IN2 := %stringValue%);
        F_EQ_Bool_WSTRING : F_EQ(IN2 := %wstringValue%);
        TIMEType : TEST_CONDITION;
      END_FBS
      EVENT_CONNECTIONS
        F_EQ_Bool.CNF TO BollType.REQ;
        F_EQ_SINT.CNF TO SINTType.REQ;
        F_EQ_INT.CNF TO INTType.REQ;
        F_EQ_DINT.CNF TO DINType.REQ;
        F_EQ_UINT.CNF TO UINTType.REQ;
        F_EQ_UDINT.CNF TO UDINTType.REQ;
        F_EQ_USINT.CNF TO USINTType.REQ;
        F_EQ_LINT.CNF TO LINTType.REQ;
        F_EQ_WORD.CNF TO WORDType.REQ;
        F_EQ_DWORD.CNF TO DWORDType.REQ;
        F_EQ_BYTE.CNF TO BYTEType.REQ;
        F_EQ_ULINT.CNF TO ULINTType.REQ;
        F_EQ_REAL.CNF TO REALType.REQ;
        F_EQ_TOD.CNF TO TODType.REQ;
        F_EQ_Bool_STRING.CNF TO STRINGType.REQ;
        F_EQ_LREAL.CNF TO LREALType.REQ;
        F_EQ_DT.CNF TO DTType.REQ;
        F_EQ_Bool_WSTRING.CNF TO WSTRINGType.REQ;
        F_EQ_LWORD.CNF TO LWORDType.REQ;
        F_EQ_DATE.CNF TO DATEType.REQ;
        F_EQ_TIME.CNF TO TIMEType.REQ;
        REQ TO F_EQ_Bool.REQ;
        BollType.CNF TO F_EQ_SINT.REQ;
        SINTType.CNF TO F_EQ_INT.REQ;
        INTType.CNF TO F_EQ_DINT.REQ;
        DINType.CNF TO F_EQ_LINT.REQ;
        LINTType.CNF TO F_EQ_USINT.REQ;
        USINTType.CNF TO F_EQ_UINT.REQ;
        UINTType.CNF TO F_EQ_UDINT.REQ;
        UDINTType.CNF TO F_EQ_ULINT.REQ;
        ULINTType.CNF TO F_EQ_BYTE.REQ;
        BYTEType.CNF TO F_EQ_WORD.REQ;
        WORDType.CNF TO F_EQ_DWORD.REQ;
        DWORDType.CNF TO F_EQ_LWORD.REQ;
        DATEType.CNF TO F_EQ_TOD.REQ;
        TODType.CNF TO F_EQ_DT.REQ;
        DTType.CNF TO F_EQ_TIME.REQ;
        TIMEType.CNF TO F_EQ_REAL.REQ;
        REALType.CNF TO F_EQ_LREAL.REQ;
        LREALType.CNF TO F_EQ_Bool_STRING.REQ;
        STRINGType.CNF TO F_EQ_Bool_WSTRING.REQ;
        LWORDType.CNF TO F_EQ_REAL.REQ;
        WSTRINGType.CNF TO CNF;
      END_CONNECTIONS
      DATA_CONNECTIONS
        F_EQ_Bool.OUT TO BollType.check;
        F_EQ_SINT.OUT TO SINTType.check;
        F_EQ_INT.OUT TO INTType.check;
        F_EQ_DINT.OUT TO DINType.check;
        F_EQ_UINT.OUT TO UINTType.check;
        F_EQ_LINT.OUT TO LINTType.check;
        F_EQ_USINT.OUT TO USINTType.check;
        F_EQ_UDINT.OUT TO UDINTType.check;
        F_EQ_WORD.OUT TO WORDType.check;
        F_EQ_ULINT.OUT TO ULINTType.check;
        F_EQ_BYTE.OUT TO BYTEType.check;
        F_EQ_DWORD.OUT TO DWORDType.check;
        F_EQ_TOD.OUT TO TODType.check;
        F_EQ_LWORD.OUT TO LWORDType.check;
        F_EQ_Bool_WSTRING.OUT TO WSTRINGType.check;
        F_EQ_LREAL.OUT TO LREALType.check;
        F_EQ_DATE.OUT TO DATEType.check;
        F_EQ_Bool_STRING.OUT TO STRINGType.check;
        F_EQ_TIME.OUT TO TIMEType.check;
        F_EQ_REAL.OUT TO REALType.check;
        F_EQ_DT.OUT TO DTType.check;
        SINT_I TO F_EQ_SINT.IN1;
        INT_I TO F_EQ_INT.IN1;
        DINT_I TO F_EQ_DINT.IN1;
        LINT_I TO F_EQ_LINT.IN1;
        USINT_I TO F_EQ_USINT.IN1;
        UINT_I TO F_EQ_UINT.IN1;
        UDINT_I TO F_EQ_UDINT.IN1;
        ULINT_I TO F_EQ_ULINT.IN1;
        BYTE_I TO F_EQ_BYTE.IN1;
        WORD_I TO F_EQ_WORD.IN1;
        DWORD_I TO F_EQ_DWORD.IN1;
        LWORD_I TO F_EQ_LWORD.IN1;
        DATE_I TO F_EQ_DATE.IN1;
        TIME_OF_DAY_I TO F_EQ_TOD.IN1;
        DATE_AND_TIME_I TO F_EQ_DT.IN1;
        TIME_I TO F_EQ_TIME.IN1;
        REAL_I TO F_EQ_REAL.IN1;
        LREAL_I TO F_EQ_LREAL.IN1;
        STRING_I TO F_EQ_Bool_STRING.IN1;
        WSTRING_I TO F_EQ_Bool_WSTRING.IN1;
        BOOL_I TO F_EQ_Bool.IN1;
      END_CONNECTIONS
    END_SUBAPPLICATION
    SUBAPPLICATION AllTypes_3
      EVENT_INPUT
        REQ;
      END_EVENT
      EVENT_OUTPUT
        CNF;
      END_EVENT
      VAR_INPUT
        BOOL_I : BOOL; (* BOOL Type Input *)
        SINT_I : SINT; (* SINT Type Input *)
        INT_I : INT; (* INT Type Input *)
        DINT_I : DINT; (* DINT Type Input *)
        LINT_I : LINT; (* LINT Type Input *)
        USINT_I : USINT; (* USINT Type Input *)
        UINT_I : UINT; (* UINT Type Input *)
        UDINT_I : UDINT; (* UDINT Type Input *)
        ULINT_I : ULINT; (* ULINT Type Input *)
        BYTE_I : BYTE; (* BYTE Type Input *)
        WORD_I : WORD; (* WORD Type Input *)
        DWORD_I : DWORD; (* DWORD Type Input *)
        LWORD_I : LWORD; (* LWORD Type Input *)
        DATE_I_BOOL : BOOL; (* DATE Type Input *)
        TIME_OF_DAY_I_BOOL : BOOL; (* TIME_OF_DAY Type Input *)
        DATE_AND_TIME_I_BOOL : BOOL; (* DATE_AND_TIME Type Input *)
        TIME_I : TIME; (* TIME Type Input *)
        REAL_I : REAL; (* REAL Type Input *)
        LREAL_I : LREAL; (* LREAL Type Input *)
        STRING_I : STRING; (* STRING Type Input *)
        WSTRING_I : WSTRING; (* WSTRING Type Input *)
      END_VAR
      VAR_OUTPUT
        BOOL_O : BOOL; (* BOOL Type Output *)
        SINT_O : SINT; (* SINT Type Output *)
        INT_O : INT; (* INT Type Output *)
        DINT_O : DINT; (* DINT Type Output *)
        LINT_O : LINT; (* LINT Type Output *)
        USINT_O : USINT; (* USINT Type Output *)
        UINT_O : UINT; (* UINT Type Output *)
        UDINT_O : UDINT; (* UDINT Type Output *)
        ULINT_O : ULINT; (* ULINT Type Output *)
        BYTE_O : BYTE; (* BYTE Type Output *)
        WORD_O : WORD; (* WORD Type Output *)
        DWORD_O : DWORD; (* DWORD Type Output *)
        LWORD_O : LWORD; (* LWORD Type Output *)
        DATE_O_BOOL : BOOL; (* DATE Type Output *)
        TIME_OF_DAY_O_BOOL : BOOL; (* TIME_OF_DAY Type Output *)
        DATE_AND_TIME_O_BOOL : BOOL; (* DATE_AND_TIME Type Output *)
        TIME_O : TIME; (* TIME Type Output *)
        REAL_O : REAL; (* REAL Type Output *)
        LREAL_O : LREAL; (* LREAL Type Output *)
        STRING_O : STRING; (* STRING Type Output *)
        WSTRING_O : WSTRING; (* WSTRING Type Output *)
      END_VAR
      FBS
        SINT2SINT : SINT2SINT;
        UINT2UINT : UINT2UINT;
        BOOL2BOOL : BOOL2BOOL;
        UDINT2UDINT : UDINT2UDINT;
        DINT2DINT : DINT2DINT;
        F_LINT_TO_INT : F_LINT_TO_INT;
        INT2INT : INT2INT;
        USINT2USINT : USINT2USINT;
        F_ULINT_TO_INT : F_ULINT_TO_INT;
        BYTE2BYTE : BYTE2BYTE;
        WORD2WORD : WORD2WORD;
        DWORD2DWORD : DWORD2DWORD;
        F_LWORD_TO_INT : F_LWORD_TO_INT;
        MISSING_DATE : F_DT_TO_DATE;
        MISSING_DATE_AND_TIME : F_DT_TO_TOD;
        TIME2TIME : TIME2TIME;
        REAL2REAL : REAL2REAL;
        LREAL2LREAL : LREAL2LREAL;
        STRING2STRING : STRING2STRING;
        WSTRING2WSTRING : WSTRING2WSTRING;
        Time_of_day : F_ADD_TOD_TIME;
        F_INT_TO_LINT : F_INT_TO_LINT;
        F_INT_TO_ULINT : F_INT_TO_ULINT;
        F_INT_TO_LWORD : F_INT_TO_LWORD;
        BOOL2BOOL_1 : BOOL2BOOL;
        BOOL2BOOL_2 : BOOL2BOOL;
        BOOL2BOOL_3 : BOOL2BOOL;
      END_FBS
      EVENT_CONNECTIONS
        REQ TO BOOL2BOOL.REQ;
        F_LINT_TO_INT.CNF TO F_INT_TO_LINT.REQ;
        F_ULINT_TO_INT.CNF TO F_INT_TO_ULINT.REQ;
        F_LWORD_TO_INT.CNF TO F_INT_TO_LWORD.REQ;
        BOOL2BOOL.CNF TO SINT2SINT.REQ;
        SINT2SINT.CNF TO INT2INT.REQ;
        INT2INT.CNF TO DINT2DINT.REQ;
        DINT2DINT.CNF TO F_LINT_TO_INT.REQ;
        F_INT_TO_LINT.CNF TO USINT2USINT.REQ;
        USINT2USINT.CNF TO UINT2UINT.REQ;
        UINT2UINT.CNF TO UDINT2UDINT.REQ;
        UDINT2UDINT.CNF TO F_ULINT_TO_INT.REQ;
        F_INT_TO_ULINT.CNF TO BYTE2BYTE.REQ;
        BYTE2BYTE.CNF TO WORD2WORD.REQ;
        WORD2WORD.CNF TO DWORD2DWORD.REQ;
        DWORD2DWORD.CNF TO F_LWORD_TO_INT.REQ;
        F_INT_TO_LWORD.CNF TO BOOL2BOOL_1.REQ;
        BOOL2BOOL_1.CNF TO BOOL2BOOL_2.REQ;
        BOOL2BOOL_2.CNF TO BOOL2BOOL_3.REQ;
        BOOL2BOOL_3.CNF TO TIME2TIME.REQ;
        TIME2TIME.CNF TO REAL2REAL.REQ;
        REAL2REAL.CNF TO LREAL2LREAL.REQ;
        LREAL2LREAL.CNF TO STRING2STRING.REQ;
        STRING2STRING.CNF TO WSTRING2WSTRING.REQ;
        WSTRING2WSTRING.CNF TO CNF;
      END_CONNECTIONS
      DATA_CONNECTIONS
        BOOL_I TO BOOL2BOOL.IN;
        SINT_I TO SINT2SINT.IN;
        INT_I TO INT2INT.IN;
        DINT_I TO DINT2DINT.IN;
        LINT_I TO F_LINT_TO_INT.IN;
        USINT_I TO USINT2USINT.IN;
        UINT_I TO UINT2UINT.IN;
        UDINT_I TO UDINT2UDINT.IN;
        ULINT_I TO F_ULINT_TO_INT.IN;
        BYTE_I TO BYTE2BYTE.IN;
        WORD_I TO WORD2WORD.IN;
        DWORD_I TO DWORD2DWORD.IN;
        LWORD_I TO F_LWORD_TO_INT.IN;
        TIME_I TO TIME2TIME.IN;
        REAL_I TO REAL2REAL.IN;
        LREAL_I TO LREAL2LREAL.IN;
        STRING_I TO STRING2STRING.IN;
        WSTRING_I TO WSTRING2WSTRING.IN;
        SINT2SINT.OUT TO SINT_O;
        INT2INT.OUT TO INT_O;
        DINT2DINT.OUT TO DINT_O;
        F_LINT_TO_INT.OUT TO F_INT_TO_LINT.IN;
        F_INT_TO_LINT.OUT TO LINT_O;
        USINT2USINT.OUT TO USINT_O;
        UINT2UINT.OUT TO UINT_O;
        UDINT2UDINT.OUT TO UDINT_O;
        F_ULINT_TO_INT.OUT TO F_INT_TO_ULINT.IN;
        F_INT_TO_ULINT.OUT TO ULINT_O;
        BYTE2BYTE.OUT TO BYTE_O;
        WORD2WORD.OUT TO WORD_O;
        DWORD2DWORD.OUT TO DWORD_O;
        F_LWORD_TO_INT.OUT TO F_INT_TO_LWORD.IN;
        F_INT_TO_LWORD.OUT TO LWORD_O;
        WSTRING2WSTRING.OUT TO WSTRING_O;
        STRING2STRING.OUT TO STRING_O;
        LREAL2LREAL.OUT TO LREAL_O;
        REAL2REAL.OUT TO REAL_O;
        TIME2TIME.OUT TO TIME_O;
        DATE_I_BOOL TO BOOL2BOOL_1.IN;
        TIME_OF_DAY_I_BOOL TO BOOL2BOOL_2.IN;
        DATE_AND_TIME_I_BOOL TO BOOL2BOOL_3.IN;
        BOOL2BOOL_1.OUT TO DATE_O_BOOL;
        BOOL2BOOL_2.OUT TO TIME_OF_DAY_O_BOOL;
        BOOL2BOOL_3.OUT TO DATE_AND_TIME_O_BOOL;
        BOOL2BOOL.OUT TO BOOL_O;
      END_CONNECTIONS
    END_SUBAPPLICATION
    EVENT_CONNECTIONS
      Read.IND TO AllTypes.REQ;
      AllTypes.CNF TO TypeTest.REQ;
      AllTypes_1.CNF TO TypeTest_1.REQ;
      Method.IND TO AllTypes_1.REQ;
      TypeTest_1.CNF TO Method.RSP;
      SUBSCRIBE_0_1.IND TO E_SR.R;
      SUBSCRIBE_0_1.INITO TO E_SR.S;
      LocalWrite.INITO TO Read.INIT;
      Read.INITO TO Method.INIT;
      E_SR.EO TO LocalWrite.INIT;
      Method.INITO TO E_SWITCH.EI;
      E_SWITCH.EO0 TO HandleInitLocal.InitFinished;
      LocalWrite.CNF TO E_DELAY.START;
      E_DELAY.EO TO HandleInitLocal.InitFinished;
      PUBLISH_0.CNF TO E_SR_2.S;
      E_PERMIT.EO TO E_SR_1.S;
      E_SR_2.EO TO E_PERMIT.EI;
      InitFinishedSignal.IND TO PUBLISH_0.REQ;
      InitFinishedSignal.INITO TO PUBLISH_0.INIT;
      RemoteRead.INITO TO RemoteCall.INIT;
      RemoteCall.INITO TO HandleInit.InitFinished;
      HandleInit.Execute TO SubApp.REQ;
      RemoteRead.CNF TO AllTypes_2.REQ;
      AllTypes_2.CNF TO TypeTest_2.REQ;
      SubApp_1.CNF TO LocalWrite.REQ;
      E_SWITCH.EO1 TO SubApp_1.REQ;
      TypeTest_3.CNF TO E_SR_1.R;
      TypeTest_2.CNF TO SubApp_2.REQ;
      SubApp_2.CNF TO RemoteCall.REQ;
      RemoteCall.CNF TO AllTypes_3.REQ;
      AllTypes_3.CNF TO TypeTest_3.REQ;
      E_SR_1.EO TO RemoteWrite.INIT;
      SubApp.CNF TO RemoteWrite.REQ;
      RemoteWrite.INITO TO RemoteRead.INIT;
      RemoteWriteAll.CNF TO RemoteRead.REQ;
      RemoteWrite.CNF TO RemoteWriteAll.REQ;
    END_CONNECTIONS
    DATA_CONNECTIONS
      Read.RD_1 TO AllTypes.BOOL_I;
      Read.RD_2 TO AllTypes.SINT_I;
      Read.RD_3 TO AllTypes.INT_I;
      Read.RD_4 TO AllTypes.DINT_I;
      Read.RD_5 TO AllTypes.LINT_I;
      Read.RD_6 TO AllTypes.USINT_I;
      Read.RD_7 TO AllTypes.UINT_I;
      Read.RD_8 TO AllTypes.UDINT_I;
      Read.RD_9 TO AllTypes.ULINT_I;
      Read.RD_10 TO AllTypes.BYTE_I;
      Read.RD_11 TO AllTypes.WORD_I;
      Read.RD_12 TO AllTypes.DWORD_I;
      Read.RD_13 TO AllTypes.LWORD_I;
      Read.RD_14 TO AllTypes.DATE_I_BOOL;
      Read.RD_15 TO AllTypes.TIME_OF_DAY_I_BOOL;
      Read.RD_16 TO AllTypes.DATE_AND_TIME_I_BOOL;
      Read.RD_17 TO AllTypes.TIME_I;
      Read.RD_18 TO AllTypes.REAL_I;
      Read.RD_19 TO AllTypes.LREAL_I;
      Read.RD_20 TO AllTypes.STRING_I;
      Read.RD_21 TO AllTypes.WSTRING_I;
      AllTypes.BOOL_O TO TypeTest.BOOL_I;
      AllTypes.SINT_O TO TypeTest.SINT_I;
      AllTypes.INT_O TO TypeTest.INT_I;
      AllTypes.DINT_O TO TypeTest.DINT_I;
      AllTypes.LINT_O TO TypeTest.LINT_I;
      AllTypes.USINT_O TO TypeTest.USINT_I;
      AllTypes.UINT_O TO TypeTest.UINT_I;
      AllTypes.UDINT_O TO TypeTest.UDINT_I;
      AllTypes.ULINT_O TO TypeTest.ULINT_I;
      AllTypes.BYTE_O TO TypeTest.BYTE_I;
      AllTypes.WORD_O TO TypeTest.WORD_I;
      AllTypes.DWORD_O TO TypeTest.DWORD_I;
      AllTypes.LWORD_O TO TypeTest.LWORD_I;
      AllTypes.DATE_O_BOOL TO TypeTest.DATE_I;
      AllTypes.TIME_OF_DAY_O_BOOL TO TypeTest.TIME_OF_DAY_I;
      AllTypes.DATE_AND_TIME_O_BOOL TO TypeTest.DATE_AND_TIME_I;
      AllTypes.TIME_O TO TypeTest.TIME_I;
      AllTypes.REAL_O TO TypeTest.REAL_I;
      AllTypes.LREAL_O TO TypeTest.LREAL_I;
      AllTypes.STRING_O TO TypeTest.STRING_I;
      AllTypes.WSTRING_O TO TypeTest.WSTRING_I;
      AllTypes_1.BOOL_O TO TypeTest_1.BOOL_I;
      AllTypes_1.SINT_O TO TypeTest_1.SINT_I;
      AllTypes_1.INT_O TO TypeTest_1.INT_I;
      AllTypes_1.DINT_O TO TypeTest_1.DINT_I;
      AllTypes_1.LINT_O TO TypeTest_1.LINT_I;
      AllTypes_1.USINT_O TO TypeTest_1.USINT_I;
      AllTypes_1.UINT_O TO TypeTest_1.UINT_I;
      AllTypes_1.UDINT_O TO TypeTest_1.UDINT_I;
      AllTypes_1.ULINT_O TO TypeTest_1.ULINT_I;
      AllTypes_1.BYTE_O TO TypeTest_1.BYTE_I;
      AllTypes_1.WORD_O TO TypeTest_1.WORD_I;
      AllTypes_1.DWORD_O TO TypeTest_1.DWORD_I;
      AllTypes_1.LWORD_O TO TypeTest_1.LWORD_I;
      AllTypes_1.DATE_O_BOOL TO TypeTest_1.DATE_I;
      AllTypes_1.TIME_OF_DAY_O_BOOL TO TypeTest_1.TIME_OF_DAY_I;
      AllTypes_1.DATE_AND_TIME_O_BOOL TO TypeTest_1.DATE_AND_TIME_I;
      AllTypes_1.TIME_O TO TypeTest_1.TIME_I;
      AllTypes_1.REAL_O TO TypeTest_1.REAL_I;
      AllTypes_1.LREAL_O TO TypeTest_1.LREAL_I;
      AllTypes_1.STRING_O TO TypeTest_1.STRING_I;
      AllTypes_1.WSTRING_O TO TypeTest_1.WSTRING_I;
      Method.RD_6 TO AllTypes_1.USINT_I;
      Method.RD_10 TO AllTypes_1.BYTE_I;
      Method.RD_18 TO AllTypes_1.REAL_I;
      Method.RD_16 TO AllTypes_1.DATE_AND_TIME_I_BOOL;
      Method.RD_11 TO AllTypes_1.WORD_I;
      Method.RD_21 TO AllTypes_1.WSTRING_I;
      Method.RD_8 TO AllTypes_1.UDINT_I;
      Method.RD_4 TO AllTypes_1.DINT_I;
      Method.RD_1 TO AllTypes_1.BOOL_I;
      Method.RD_17 TO AllTypes_1.TIME_I;
      Method.RD_3 TO AllTypes_1.INT_I;
      Method.RD_20 TO AllTypes_1.STRING_I;
      Method.RD_13 TO AllTypes_1.LWORD_I;
      Method.RD_5 TO AllTypes_1.LINT_I;
      Method.RD_12 TO AllTypes_1.DWORD_I;
      Method.RD_7 TO AllTypes_1.UINT_I;
      Method.RD_2 TO AllTypes_1.SINT_I;
      Method.RD_9 TO AllTypes_1.ULINT_I;
      Method.RD_14 TO AllTypes_1.DATE_I_BOOL;
      Method.RD_19 TO AllTypes_1.LREAL_I;
      Method.RD_15 TO AllTypes_1.TIME_OF_DAY_I_BOOL;
      AllTypes_1.BOOL_O TO Method.SD_1;
      AllTypes_1.SINT_O TO Method.SD_2;
      AllTypes_1.INT_O TO Method.SD_3;
      AllTypes_1.DINT_O TO Method.SD_4;
      AllTypes_1.LINT_O TO Method.SD_5;
      AllTypes_1.USINT_O TO Method.SD_6;
      AllTypes_1.UINT_O TO Method.SD_7;
      AllTypes_1.UDINT_O TO Method.SD_8;
      AllTypes_1.ULINT_O TO Method.SD_9;
      AllTypes_1.BYTE_O TO Method.SD_10;
      AllTypes_1.WORD_O TO Method.SD_11;
      AllTypes_1.DWORD_O TO Method.SD_12;
      AllTypes_1.LWORD_O TO Method.SD_13;
      AllTypes_1.DATE_O_BOOL TO Method.SD_14;
      AllTypes_1.TIME_OF_DAY_O_BOOL TO Method.SD_15;
      AllTypes_1.DATE_AND_TIME_O_BOOL TO Method.SD_16;
      AllTypes_1.TIME_O TO Method.SD_17;
      AllTypes_1.REAL_O TO Method.SD_18;
      AllTypes_1.LREAL_O TO Method.SD_19;
      AllTypes_1.STRING_O TO Method.SD_20;
      AllTypes_1.WSTRING_O TO Method.SD_21;
      Method.RD_1 TO AllTypes_1.BOOL_I;
      Method.RD_2 TO AllTypes_1.SINT_I;
      Method.RD_3 TO AllTypes_1.INT_I;
      Method.RD_4 TO AllTypes_1.DINT_I;
      Method.RD_5 TO AllTypes_1.LINT_I;
      Method.RD_6 TO AllTypes_1.USINT_I;
      Method.RD_7 TO AllTypes_1.UINT_I;
      Method.RD_8 TO AllTypes_1.UDINT_I;
      Method.RD_9 TO AllTypes_1.ULINT_I;
      Method.RD_10 TO AllTypes_1.BYTE_I;
      Method.RD_11 TO AllTypes_1.WORD_I;
      Method.RD_12 TO AllTypes_1.DWORD_I;
      Method.RD_13 TO AllTypes_1.LWORD_I;
      Method.RD_14 TO AllTypes_1.DATE_I_BOOL;
      Method.RD_15 TO AllTypes_1.TIME_OF_DAY_I_BOOL;
      Method.RD_16 TO AllTypes_1.DATE_AND_TIME_I_BOOL;
      Method.RD_17 TO AllTypes_1.TIME_I;
      Method.RD_18 TO AllTypes_1.REAL_I;
      Method.RD_19 TO AllTypes_1.LREAL_I;
      Method.RD_20 TO AllTypes_1.STRING_I;
      Method.RD_21 TO AllTypes_1.WSTRING_I;
      Read.RD_1 TO AllTypes.BOOL_I;
      Read.RD_2 TO AllTypes.SINT_I;
      Read.RD_3 TO AllTypes.INT_I;
      Read.RD_4 TO AllTypes.DINT_I;
      Read.RD_5 TO AllTypes.LINT_I;
      Read.RD_6 TO AllTypes.USINT_I;
      Read.RD_7 TO AllTypes.UINT_I;
      Read.RD_8 TO AllTypes.UDINT_I;
      Read.RD_9 TO AllTypes.ULINT_I;
      Read.RD_10 TO AllTypes.BYTE_I;
      Read.RD_11 TO AllTypes.WORD_I;
      Read.RD_12 TO AllTypes.DWORD_I;
      Read.RD_13 TO AllTypes.LWORD_I;
      Read.RD_14 TO AllTypes.DATE_I_BOOL;
      Read.RD_15 TO AllTypes.TIME_OF_DAY_I_BOOL;
      Read.RD_16 TO AllTypes.DATE_AND_TIME_I_BOOL;
      Read.RD_17 TO AllTypes.TIME_I;
      Read.RD_18 TO AllTypes.REAL_I;
      Read.RD_19 TO AllTypes.LREAL_I;
      Read.RD_20 TO AllTypes.STRING_I;
      Read.RD_21 TO AllTypes.WSTRING_I;
      AllTypes_2.BOOL_O TO TypeTest_2.BOOL_I;
      AllTypes_2.SINT_O TO TypeTest_2.SINT_I;
      AllTypes_2.INT_O TO TypeTest_2.INT_I;
      AllTypes_2.DINT_O TO TypeTest_2.DINT_I;
      AllTypes_2.LINT_O TO TypeTest_2.LINT_I;
      AllTypes_2.USINT_O TO TypeTest_2.USINT_I;
      AllTypes_2.UINT_O TO TypeTest_2.UINT_I;
      AllTypes_2.UDINT_O TO TypeTest_2.UDINT_I;
      AllTypes_2.ULINT_O TO TypeTest_2.ULINT_I;
      AllTypes_2.BYTE_O TO TypeTest_2.BYTE_I;
      AllTypes_2.WORD_O TO TypeTest_2.WORD_I;
      AllTypes_2.DWORD_O TO TypeTest_2.DWORD_I;
      AllTypes_2.LWORD_O TO TypeTest_2.LWORD_I;
      AllTypes_2.DATE_O_BOOL TO TypeTest_2.DATE_I;
      AllTypes_2.TIME_OF_DAY_O_BOOL TO TypeTest_2.TIME_OF_DAY_I;
      AllTypes_2.DATE_AND_TIME_O_BOOL TO TypeTest_2.DATE_AND_TIME_I;
      AllTypes_2.TIME_O TO TypeTest_2.TIME_I;
      AllTypes_2.REAL_O TO TypeTest_2.REAL_I;
      AllTypes_2.LREAL_O TO TypeTest_2.LREAL_I;
      AllTypes_2.STRING_O TO TypeTest_2.STRING_I;
      AllTypes_2.WSTRING_O TO TypeTest_2.WSTRING_I;
      AllTypes_3.BOOL_O TO TypeTest_3.BOOL_I;
      AllTypes_3.SINT_O TO TypeTest_3.SINT_I;
      AllTypes_3.INT_O TO TypeTest_3.INT_I;
      AllTypes_3.DINT_O TO TypeTest_3.DINT_I;
      AllTypes_3.LINT_O TO TypeTest_3.LINT_I;
      AllTypes_3.USINT_O TO TypeTest_3.USINT_I;
      AllTypes_3.UINT_O TO TypeTest_3.UINT_I;
      AllTypes_3.UDINT_O TO TypeTest_3.UDINT_I;
      AllTypes_3.ULINT_O TO TypeTest_3.ULINT_I;
      AllTypes_3.BYTE_O TO TypeTest_3.BYTE_I;
      AllTypes_3.WORD_O TO TypeTest_3.WORD_I;
      AllTypes_3.DWORD_O TO TypeTest_3.DWORD_I;
      AllTypes_3.LWORD_O TO TypeTest_3.LWORD_I;
      AllTypes_3.DATE_O_BOOL TO TypeTest_3.DATE_I;
      AllTypes_3.TIME_OF_DAY_O_BOOL TO TypeTest_3.TIME_OF_DAY_I;
      AllTypes_3.DATE_AND_TIME_O_BOOL TO TypeTest_3.DATE_AND_TIME_I;
      AllTypes_3.TIME_O TO TypeTest_3.TIME_I;
      AllTypes_3.REAL_O TO TypeTest_3.REAL_I;
      AllTypes_3.LREAL_O TO TypeTest_3.LREAL_I;
      AllTypes_3.STRING_O TO TypeTest_3.STRING_I;
      AllTypes_3.WSTRING_O TO TypeTest_3.WSTRING_I;
      E_SR.Q TO HandleInitLocal.QI;
      E_SR.Q TO LocalWrite.QI;
      E_SR.Q TO Read.QI;
      E_SR.Q TO Method.QI;
      E_SR.Q TO E_SWITCH.G;
      E_SR_2.Q TO E_PERMIT.PERMIT;
      E_SR_1.Q TO HandleInit.QI;
      E_SR_1.Q TO RemoteRead.QI;
      E_SR_1.Q TO RemoteCall.QI;
      RemoteRead.RD_1 TO AllTypes_2.BOOL_I;
      RemoteRead.RD_2 TO AllTypes_2.SINT_I;
      RemoteRead.RD_3 TO AllTypes_2.INT_I;
      RemoteRead.RD_4 TO AllTypes_2.DINT_I;
      RemoteRead.RD_5 TO AllTypes_2.LINT_I;
      RemoteRead.RD_6 TO AllTypes_2.USINT_I;
      RemoteRead.RD_7 TO AllTypes_2.UINT_I;
      RemoteRead.RD_8 TO AllTypes_2.UDINT_I;
      RemoteRead.RD_9 TO AllTypes_2.ULINT_I;
      RemoteRead.RD_10 TO AllTypes_2.BYTE_I;
      RemoteRead.RD_11 TO AllTypes_2.WORD_I;
      RemoteRead.RD_12 TO AllTypes_2.DWORD_I;
      RemoteRead.RD_13 TO AllTypes_2.LWORD_I;
      RemoteRead.RD_14 TO AllTypes_2.DATE_I_BOOL;
      RemoteRead.RD_15 TO AllTypes_2.TIME_OF_DAY_I_BOOL;
      RemoteRead.RD_16 TO AllTypes_2.DATE_AND_TIME_I_BOOL;
      RemoteRead.RD_17 TO AllTypes_2.TIME_I;
      RemoteRead.RD_18 TO AllTypes_2.REAL_I;
      RemoteRead.RD_19 TO AllTypes_2.LREAL_I;
      RemoteRead.RD_20 TO AllTypes_2.STRING_I;
      RemoteRead.RD_21 TO AllTypes_2.WSTRING_I;
      SubApp_1.BOOL_O TO LocalWrite.SD_1;
      SubApp_1.SINT_O TO LocalWrite.SD_2;
      SubApp_1.INT_O TO LocalWrite.SD_3;
      SubApp_1.DINT_O TO LocalWrite.SD_4;
      SubApp_1.LINT_O TO LocalWrite.SD_5;
      SubApp_1.USINT_O TO LocalWrite.SD_6;
      SubApp_1.UINT_O TO LocalWrite.SD_7;
      SubApp_1.UDINT_O TO LocalWrite.SD_8;
      SubApp_1.ULINT_O TO LocalWrite.SD_9;
      SubApp_1.BYTE_O TO LocalWrite.SD_10;
      SubApp_1.WORD_O TO LocalWrite.SD_11;
      SubApp_1.DWORD_O TO LocalWrite.SD_12;
      SubApp_1.LWORD_O TO LocalWrite.SD_13;
      SubApp_1.DATE_O TO LocalWrite.SD_14;
      SubApp_1.DATE_TIME_O TO LocalWrite.SD_15;
      SubApp_1.TIME_OF_DAY_O TO LocalWrite.SD_16;
      SubApp_1.TIME_O TO LocalWrite.SD_17;
      SubApp_1.REAL_O TO LocalWrite.SD_18;
      SubApp_1.LREAL_O TO LocalWrite.SD_19;
      SubApp_1.STRING_O TO LocalWrite.SD_20;
      SubApp_1.WSTRING_O TO LocalWrite.SD_21;
      SubApp_2.BOOL_O TO RemoteCall.SD_1;
      SubApp_2.SINT_O TO RemoteCall.SD_2;
      SubApp_2.INT_O TO RemoteCall.SD_3;
      SubApp_2.DINT_O TO RemoteCall.SD_4;
      SubApp_2.LINT_O TO RemoteCall.SD_5;
      SubApp_2.USINT_O TO RemoteCall.SD_6;
      SubApp_2.UINT_O TO RemoteCall.SD_7;
      SubApp_2.UDINT_O TO RemoteCall.SD_8;
      SubApp_2.ULINT_O TO RemoteCall.SD_9;
      SubApp_2.BYTE_O TO RemoteCall.SD_10;
      SubApp_2.WORD_O TO RemoteCall.SD_11;
      SubApp_2.DWORD_O TO RemoteCall.SD_12;
      SubApp_2.LWORD_O TO RemoteCall.SD_13;
      SubApp_2.DATE_O TO RemoteCall.SD_14;
      SubApp_2.DATE_TIME_O TO RemoteCall.SD_15;
      SubApp_2.TIME_OF_DAY_O TO RemoteCall.SD_16;
      SubApp_2.TIME_O TO RemoteCall.SD_17;
      SubApp_2.REAL_O TO RemoteCall.SD_18;
      SubApp_2.LREAL_O TO RemoteCall.SD_19;
      SubApp_2.STRING_O TO RemoteCall.SD_20;
      SubApp_2.WSTRING_O TO RemoteCall.SD_21;
      RemoteCall.RD_1 TO AllTypes_3.BOOL_I;
      RemoteCall.RD_2 TO AllTypes_3.SINT_I;
      RemoteCall.RD_3 TO AllTypes_3.INT_I;
      RemoteCall.RD_4 TO AllTypes_3.DINT_I;
      RemoteCall.RD_5 TO AllTypes_3.LINT_I;
      RemoteCall.RD_6 TO AllTypes_3.USINT_I;
      RemoteCall.RD_7 TO AllTypes_3.UINT_I;
      RemoteCall.RD_8 TO AllTypes_3.UDINT_I;
      RemoteCall.RD_9 TO AllTypes_3.ULINT_I;
      RemoteCall.RD_10 TO AllTypes_3.BYTE_I;
      RemoteCall.RD_11 TO AllTypes_3.WORD_I;
      RemoteCall.RD_12 TO AllTypes_3.DWORD_I;
      RemoteCall.RD_13 TO AllTypes_3.LWORD_I;
      RemoteCall.RD_14 TO AllTypes_3.DATE_I_BOOL;
      RemoteCall.RD_15 TO AllTypes_3.TIME_OF_DAY_I_BOOL;
      RemoteCall.RD_16 TO AllTypes_3.DATE_AND_TIME_I_BOOL;
      RemoteCall.RD_17 TO AllTypes_3.TIME_I;
      RemoteCall.RD_18 TO AllTypes_3.REAL_I;
      RemoteCall.RD_19 TO AllTypes_3.LREAL_I;
      RemoteCall.RD_20 TO AllTypes_3.STRING_I;
      RemoteCall.RD_21 TO AllTypes_3.WSTRING_I;
      RemoteRead.RD_1 TO AllTypes_2.BOOL_I;
      RemoteRead.RD_2 TO AllTypes_2.SINT_I;
      RemoteRead.RD_3 TO AllTypes_2.INT_I;
      RemoteRead.RD_4 TO AllTypes_2.DINT_I;
      RemoteRead.RD_5 TO AllTypes_2.LINT_I;
      RemoteRead.RD_6 TO AllTypes_2.USINT_I;
      RemoteRead.RD_7 TO AllTypes_2.UINT_I;
      RemoteRead.RD_8 TO AllTypes_2.UDINT_I;
      RemoteRead.RD_9 TO AllTypes_2.ULINT_I;
      RemoteRead.RD_10 TO AllTypes_2.BYTE_I;
      RemoteRead.RD_11 TO AllTypes_2.WORD_I;
      RemoteRead.RD_12 TO AllTypes_2.DWORD_I;
      RemoteRead.RD_13 TO AllTypes_2.LWORD_I;
      RemoteRead.RD_14 TO AllTypes_2.DATE_I_BOOL;
      RemoteRead.RD_15 TO AllTypes_2.TIME_OF_DAY_I_BOOL;
      RemoteRead.RD_16 TO AllTypes_2.DATE_AND_TIME_I_BOOL;
      RemoteRead.RD_17 TO AllTypes_2.TIME_I;
      RemoteRead.RD_18 TO AllTypes_2.REAL_I;
      RemoteRead.RD_19 TO AllTypes_2.LREAL_I;
      RemoteRead.RD_20 TO AllTypes_2.STRING_I;
      RemoteRead.RD_21 TO AllTypes_2.WSTRING_I;
      RemoteCall.RD_1 TO AllTypes_3.BOOL_I;
      RemoteCall.RD_2 TO AllTypes_3.SINT_I;
      RemoteCall.RD_3 TO AllTypes_3.INT_I;
      RemoteCall.RD_4 TO AllTypes_3.DINT_I;
      RemoteCall.RD_5 TO AllTypes_3.LINT_I;
      RemoteCall.RD_6 TO AllTypes_3.USINT_I;
      RemoteCall.RD_7 TO AllTypes_3.UINT_I;
      RemoteCall.RD_8 TO AllTypes_3.UDINT_I;
      RemoteCall.RD_9 TO AllTypes_3.ULINT_I;
      RemoteCall.RD_10 TO AllTypes_3.BYTE_I;
      RemoteCall.RD_11 TO AllTypes_3.WORD_I;
      RemoteCall.RD_12 TO AllTypes_3.DWORD_I;
      RemoteCall.RD_13 TO AllTypes_3.LWORD_I;
      RemoteCall.RD_14 TO AllTypes_3.DATE_I_BOOL;
      RemoteCall.RD_15 TO AllTypes_3.TIME_OF_DAY_I_BOOL;
      RemoteCall.RD_16 TO AllTypes_3.DATE_AND_TIME_I_BOOL;
      RemoteCall.RD_17 TO AllTypes_3.TIME_I;
      RemoteCall.RD_18 TO AllTypes_3.REAL_I;
      RemoteCall.RD_19 TO AllTypes_3.LREAL_I;
      RemoteCall.RD_20 TO AllTypes_3.STRING_I;
      RemoteCall.RD_21 TO AllTypes_3.WSTRING_I;
      E_SR_1.Q TO HandleInit.QI;
      E_SR_1.Q TO RemoteWrite.QI;
      SubApp.BOOL_O TO RemoteWrite.SD_1;
      SubApp.SINT_O TO RemoteWrite.SD_2;
      SubApp.INT_O TO RemoteWrite.SD_3;
      SubApp.DINT_O TO RemoteWrite.SD_4;
      SubApp.LINT_O TO RemoteWrite.SD_5;
      SubApp.USINT_O TO RemoteWrite.SD_6;
      SubApp.UINT_O TO RemoteWrite.SD_7;
      SubApp.UDINT_O TO RemoteWrite.SD_8;
      SubApp.ULINT_O TO RemoteWrite.SD_9;
      SubApp.BYTE_O TO RemoteWrite.SD_10;
      SubApp.WORD_o TO RemoteWrite.SD_11;
      SubApp.DWORD_O TO RemoteWrite.SD_12;
      SubApp.LWORD_O TO RemoteWrite.SD_13;
      SubApp.DATE_O TO RemoteWrite.SD_14;
      SubApp.DATE_TIME_O TO RemoteWrite.SD_15;
      SubApp.TIME_OF_DAY_O TO RemoteWrite.SD_16;
      SubApp.TIME_O TO RemoteWrite.SD_17;
      SubApp.REAL_O TO RemoteWrite.SD_18;
      SubApp.LREAL_O TO RemoteWrite.SD_19;
      SubApp.STRING_O TO RemoteWrite.SD_20;
      SubApp.WSTRING_O TO RemoteWrite.SD_21;
      RemoteWrite.QO TO RemoteWriteAll.check;
    END_CONNECTIONS
  END_APPLICATION
  APPLICATION ShortTests
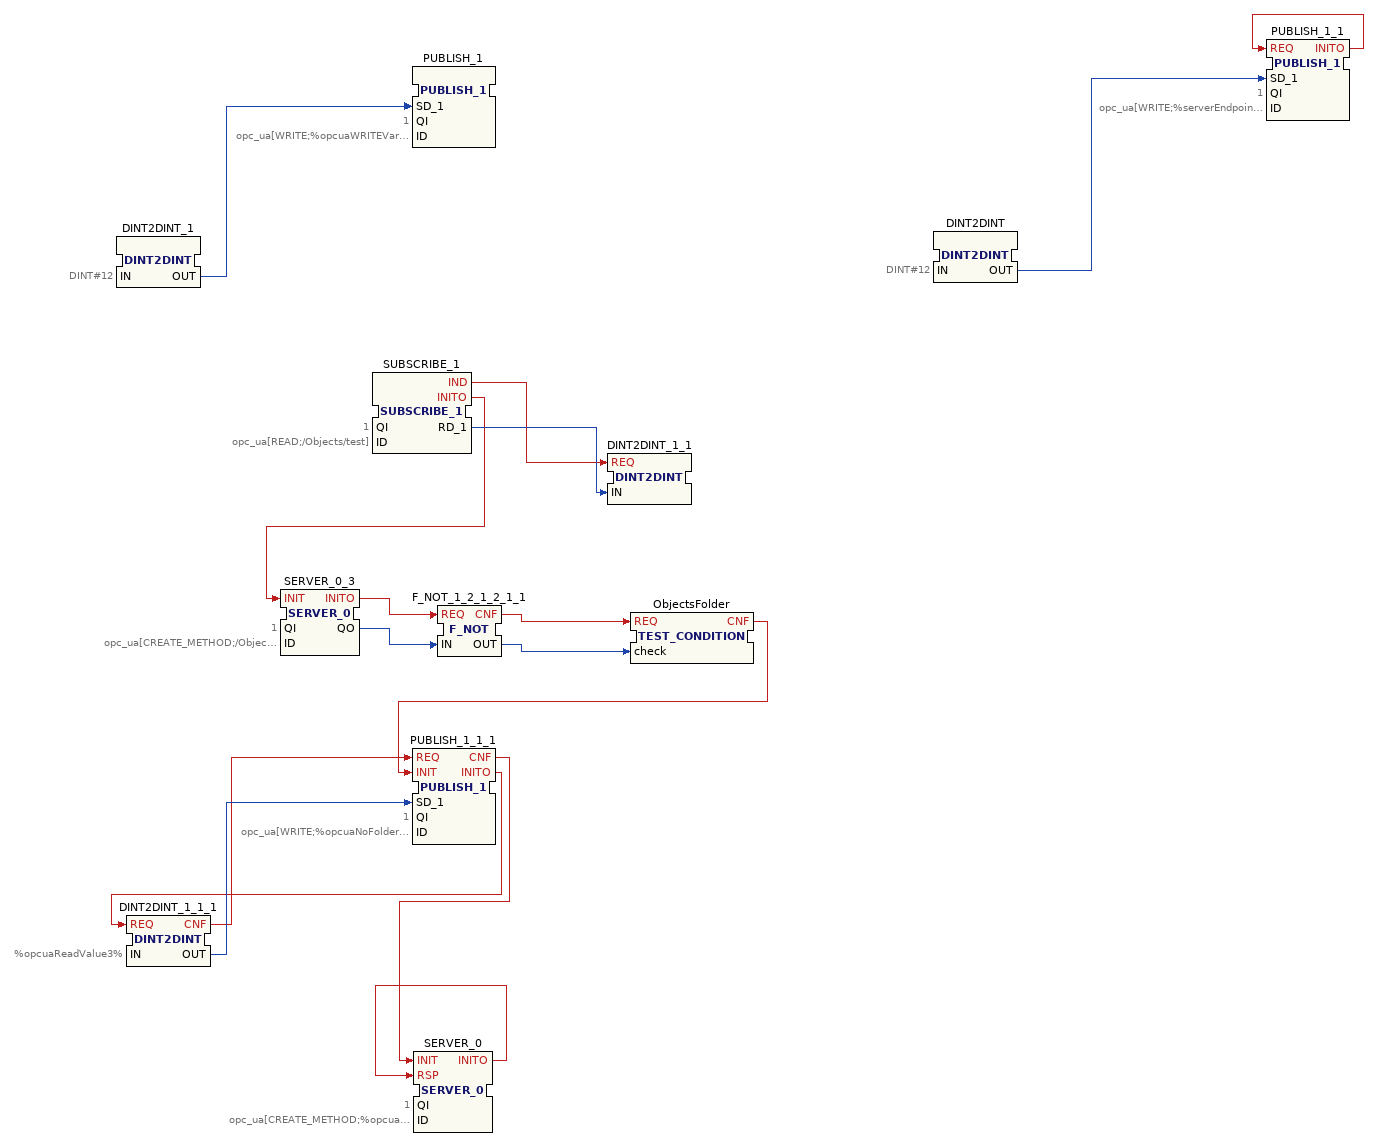
    FBS
      PUBLISH_1 : PUBLISH_1(QI := 1, ID := opc_ua[WRITE;%opcuaWRITEVariable%]);
      DINT2DINT : DINT2DINT(IN := DINT#12);
      PUBLISH_1_1 : PUBLISH_1(QI := 1, ID := opc_ua[WRITE;%serverEndpoint%;%opcuaWRITEVariable%]);
      DINT2DINT_1 : DINT2DINT(IN := DINT#12);
      SUBSCRIBE_1 : SUBSCRIBE_1(QI := 1, ID := opc_ua[READ;/Objects/test]);
      DINT2DINT_1_1 : DINT2DINT;
      ObjectsFolder : TEST_CONDITION;
      F_NOT_1_2_1_2_1_1 : F_NOT;
      SERVER_0_3 : SERVER_0(QI := 1, ID := opc_ua[CREATE_METHOD;/Objects]);
      SERVER_0 : SERVER_0(QI := 1, ID := opc_ua[CREATE_METHOD;%opcuaNoFolderMethod%]);
      DINT2DINT_1_1_1 : DINT2DINT(IN := %opcuaReadValue3%);
      PUBLISH_1_1_1 : PUBLISH_1(QI := 1, ID := opc_ua[WRITE;%opcuaNoFolder%]);
    END_FBS
    EVENT_CONNECTIONS
      PUBLISH_1_1.INITO TO PUBLISH_1_1.REQ;
      SUBSCRIBE_1.IND TO DINT2DINT_1_1.REQ;
      F_NOT_1_2_1_2_1_1.CNF TO ObjectsFolder.REQ;
      SERVER_0_3.INITO TO F_NOT_1_2_1_2_1_1.REQ;
      SUBSCRIBE_1.INITO TO SERVER_0_3.INIT;
      DINT2DINT_1_1_1.CNF TO PUBLISH_1_1_1.REQ;
      PUBLISH_1_1_1.CNF TO SERVER_0.INIT;
      ObjectsFolder.CNF TO PUBLISH_1_1_1.INIT;
      SERVER_0.INITO TO SERVER_0.RSP;
      PUBLISH_1_1_1.INITO TO DINT2DINT_1_1_1.REQ;
    END_CONNECTIONS
    DATA_CONNECTIONS
      DINT2DINT.OUT TO PUBLISH_1_1.SD_1;
      DINT2DINT_1.OUT TO PUBLISH_1.SD_1;
      SUBSCRIBE_1.RD_1 TO DINT2DINT_1_1.IN;
      SERVER_0_3.QO TO F_NOT_1_2_1_2_1_1.IN;
      F_NOT_1_2_1_2_1_1.OUT TO ObjectsFolder.check;
      DINT2DINT_1_1_1.OUT TO PUBLISH_1_1_1.SD_1;
    END_CONNECTIONS
  END_APPLICATION
  DEVICE OPCUAServer : FORTE_PC(MGR_ID := "localhost:61500")
    {SET_ATTRIBUTE(Profile, HOLOBLOC)} (* device profile *)
    RESOURCE WrongParameters : EMB_RES
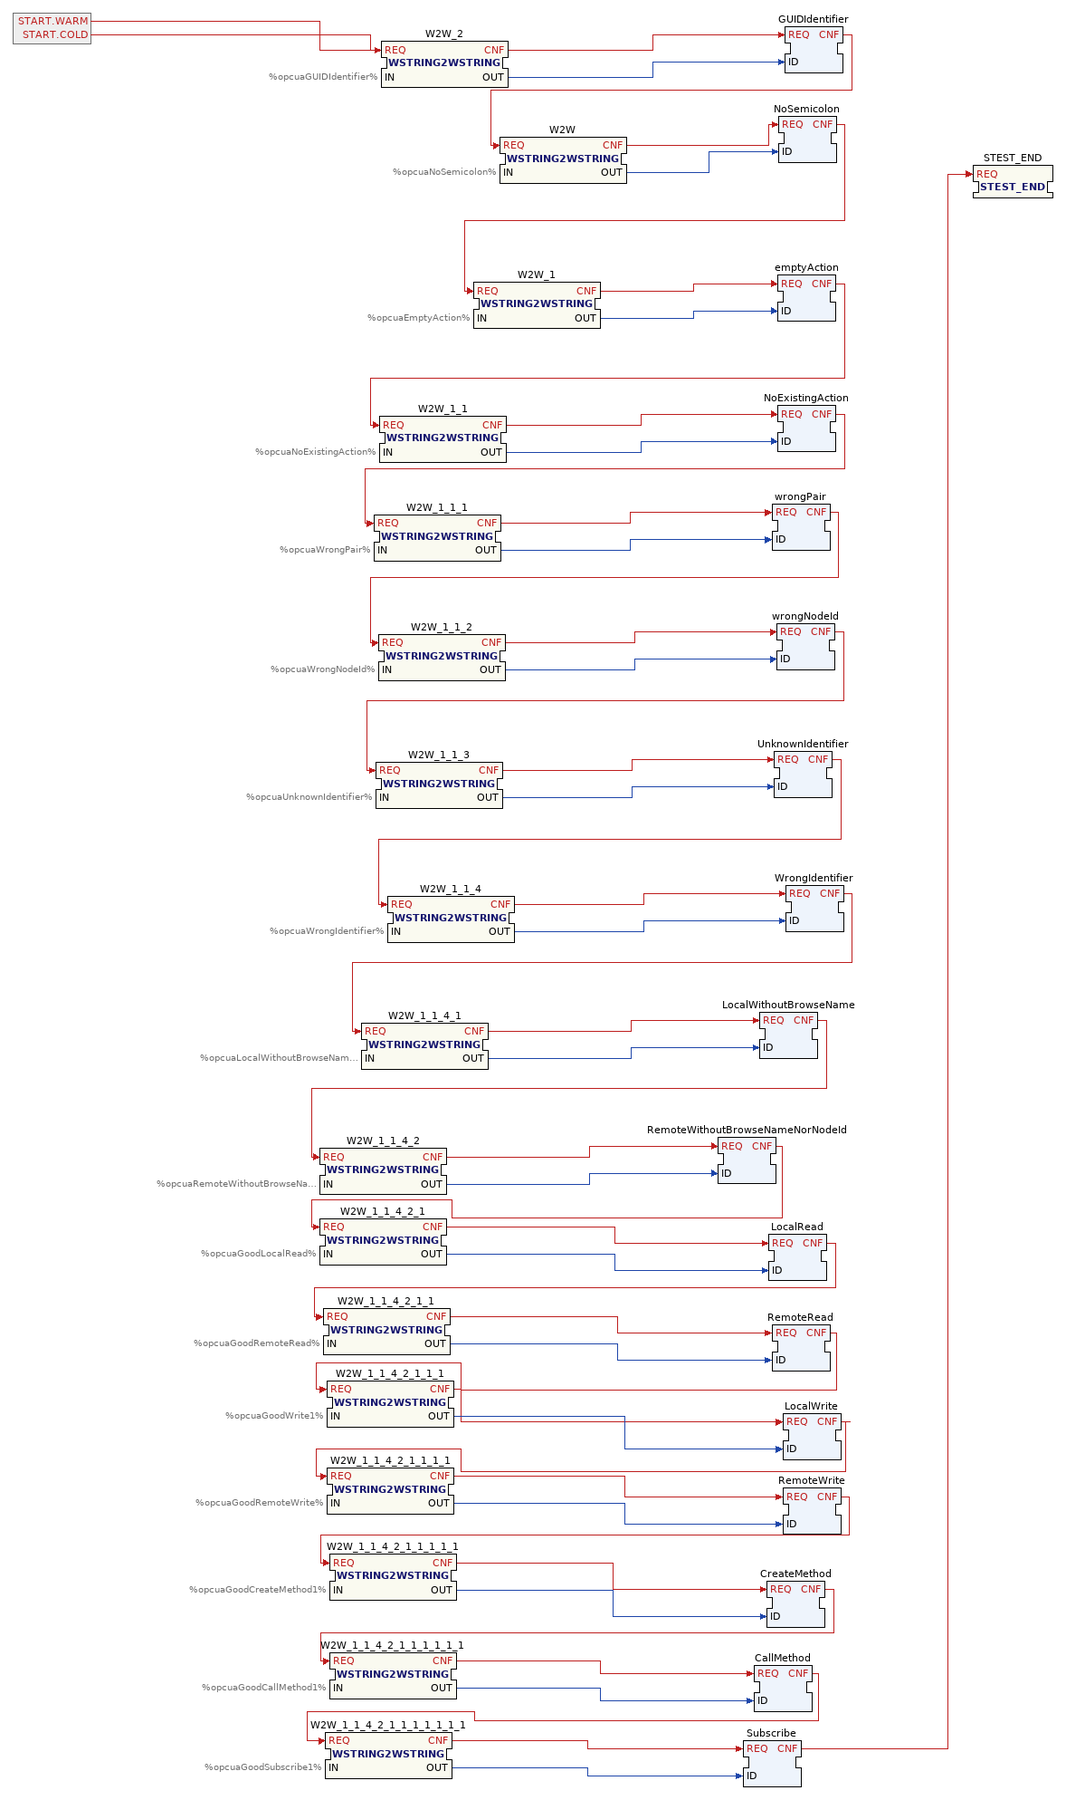
      FBS
        STEST_END : STEST_END;
        W2W : WSTRING2WSTRING(IN := %opcuaNoSemicolon%);
        W2W_1 : WSTRING2WSTRING(IN := %opcuaEmptyAction%);
        W2W_1_1 : WSTRING2WSTRING(IN := %opcuaNoExistingAction%);
        W2W_1_1_1 : WSTRING2WSTRING(IN := %opcuaWrongPair%);
        W2W_1_1_4 : WSTRING2WSTRING(IN := %opcuaWrongIdentifier%);
        W2W_1_1_2 : WSTRING2WSTRING(IN := %opcuaWrongNodeId%);
        W2W_1_1_3 : WSTRING2WSTRING(IN := %opcuaUnknownIdentifier%);
        W2W_1_1_4_1 : WSTRING2WSTRING(IN := %opcuaLocalWithoutBrowseName%);
        W2W_1_1_4_2 : WSTRING2WSTRING(IN := %opcuaRemoteWithoutBrowseNameNorNodeId%);
        W2W_1_1_4_2_1_1 : WSTRING2WSTRING(IN := %opcuaGoodRemoteRead%);
        W2W_1_1_4_2_1 : WSTRING2WSTRING(IN := %opcuaGoodLocalRead%);
        W2W_1_1_4_2_1_1_1 : WSTRING2WSTRING(IN := %opcuaGoodWrite1%);
